LIN {X 0,Y 530.457,Z 403.715,A -85,B 0,C 180,E1 -4406.963,E2 -4406.963} C_VEL
LIN {X 0,Y 530.411,Z 405.124,A -85,B 0,C 180,E1 -4407.723,E2 -4407.723} C_VEL
LIN {X 0,Y 530.344,Z 406.736,A -85,B 0,C 180,E1 -4409.242,E2 -4409.242} C_VEL
LIN {X 0,Y 530.343,Z 406.953,A -85,B 0,C 180,E1 -4410.001,E2 -4410.001} C_VEL
LIN {X 0,Y 530.344,Z 406.734,A -85,B 0,C 180,E1 -4410.76,E2 -4410.76} C_VEL
LIN {X 0,Y 530.411,Z 405.118,A -85,B 0,C 180,E1 -4412.279,E2 -4412.279} C_VEL
LIN {X 0,Y 530.457,Z 403.708,A -85,B 0,C 180,E1 -4413.039,E2 -4413.039} C_VEL
LIN {X 0,Y 530.523,Z 400.73,A -85,B 0,C 180,E1 -4414.179,E2 -4414.179} C_VEL
LIN {X 0,Y 530.525,Z 396.658,A -85,B 0,C 180,E1 -4415.322,E2 -4415.322} C_VEL
LIN {X 0,Y 530.6,Z 390.764,A -85,B 0,C 180,E1 -4416.583,E2 -4416.583} C_VEL
LIN {X 0,Y 530.729,Z 383.488,A -85,B 0,C 180,E1 -4417.802,E2 -4417.802} C_VEL
LIN {X 0,Y 530.908,Z 374.945,A -85,B 0,C 180,E1 -4418.949,E2 -4418.949} C_VEL
LIN {X 0,Y 531.113,Z 365.145,A -85,B 0,C 180,E1 -4420.003,E2 -4420.003} C_VEL
LIN {X 0,Y 531.358,Z 354.095,A -85,B 0,C 180,E1 -4420.961,E2 -4420.961} C_VEL
LIN {X 0,Y 531.545,Z 343.017,A -85,B 0,C 180,E1 -4421.73,E2 -4421.73} C_VEL
LIN {X 0,Y 531.803,Z 330.634,A -85,B 0,C 180,E1 -4422.402,E2 -4422.402} C_VEL
LIN {X 0,Y 532.021,Z 317.664,A -85,B 0,C 180,E1 -4422.93,E2 -4422.93} C_VEL
LIN {X 0,Y 532.196,Z 304.731,A -85,B 0,C 180,E1 -4423.29,E2 -4423.29} C_VEL
LIN {X 0,Y 531.121,Z 293.757,A -85,B 0,C 180,E1 -4423.512,E2 -4423.512} C_VEL
LIN {X 0,Y 531.444,Z 271.801,A -85,B 0,C 180,E1 -4426.717,E2 -4426.717} C_VEL
LIN {X 0,Y 531.874,Z 250.491,A -85,B 0,C 180,E1 -4429.893,E2 -4429.893} C_VEL
LIN {X 0,Y 532.32,Z 231.821,A -85,B 0,C 180,E1 -4432.718,E2 -4432.718} C_VEL
LIN {X 0,Y 532.927,Z 210.283,A -85,B 0,C 180,E1 -4436.036,E2 -4436.036} C_VEL
LIN {X 0,Y 533.581,Z 192.22,A -85,B 0,C 180,E1 -4438.951,E2 -4438.951} C_VEL
LIN {X 0,Y 533.493,Z 188.442,A -85,B 0,C 180,E1 -4439.604,E2 -4439.604} C_VEL
LIN {X 0,Y 530.975,Z 177.349,A -85,B 0,C 180,E1 -4441.745,E2 -4441.745} C_VEL
LIN {X 0,Y 530.961,Z 177.352,A -85,B 0,C 180,E1 -4444.849,E2 -4444.849} C_VEL
LIN {X 0,Y 530.967,Z 177.345,A -85,B 0,C 180,E1 -4447.508,E2 -4447.508} C_VEL
LIN {X 0,Y 530.982,Z 177.347,A -85,B 0,C 180,E1 -4450.434,E2 -4450.434} C_VEL
LIN {X 0,Y 530.965,Z 177.345,A -85,B 0,C 180,E1 -4453.281,E2 -4453.281} C_VEL
LIN {X 0,Y 530.981,Z 177.348,A -85,B 0,C 180,E1 -4455.623,E2 -4455.623} C_VEL
LIN {X 0,Y 530.998,Z 177.341,A -85,B 0,C 180,E1 -4458.565,E2 -4458.565} C_VEL
LIN {X 0,Y 530.956,Z 177.347,A -85,B 0,C 180,E1 -4461.529,E2 -4461.529} C_VEL
LIN {X 0,Y 530.931,Z 177.355,A -85,B 0,C 180,E1 -4464.378,E2 -4464.378} C_VEL
LIN {X 0,Y 530.931,Z 177.42,A -85,B 0,C 180,E1 -4465.823,E2 -4465.823} C_VEL
LIN {X 0,Y 530.978,Z 185.304,A -85,B 0,C 180,E1 -4468.032,E2 -4468.032} C_VEL
LIN {X 0,Y 530.976,Z 194.876,A -85,B 0,C 180,E1 -4470.878,E2 -4470.878} C_VEL
LIN {X 0,Y 531.024,Z 203.845,A -85,B 0,C 180,E1 -4473.681,E2 -4473.681} C_VEL
LIN {X 0,Y 531.011,Z 212.797,A -85,B 0,C 180,E1 -4476.606,E2 -4476.606} C_VEL
LIN {X 0,Y 530.947,Z 221.236,A -85,B 0,C 180,E1 -4479.465,E2 -4479.465} C_VEL
LIN {X 0,Y 530.848,Z 229.893,A -85,B 0,C 180,E1 -4482.407,E2 -4482.407} C_VEL
LIN {X 0,Y 530.784,Z 238.562,A -85,B 0,C 180,E1 -4485.429,E2 -4485.429} C_VEL
LIN {X 0,Y 530.747,Z 241.715,A -85,B 0,C 180,E1 -4486.552,E2 -4486.552} C_VEL
LIN {X 0,Y 532.328,Z 250.665,A -85,B 0,C 180,E1 -4486.787,E2 -4486.787} C_VEL
LIN {X 0,Y 532.167,Z 262.9,A -85,B 0,C 180,E1 -4487.172,E2 -4487.172} C_VEL
LIN {X 0,Y 531.923,Z 274.906,A -85,B 0,C 180,E1 -4487.699,E2 -4487.699} C_VEL
LIN {X 0,Y 531.711,Z 286.037,A -85,B 0,C 180,E1 -4488.337,E2 -4488.337} C_VEL
LIN {X 0,Y 531.433,Z 297.075,A -85,B 0,C 180,E1 -4489.138,E2 -4489.138} C_VEL
LIN {X 0,Y 531.198,Z 307.619,A -85,B 0,C 180,E1 -4490.096,E2 -4490.096} C_VEL
LIN {X 0,Y 531.002,Z 316.164,A -85,B 0,C 180,E1 -4491.053,E2 -4491.053} C_VEL
LIN {X 0,Y 530.785,Z 324.463,A -85,B 0,C 180,E1 -4492.2,E2 -4492.2} C_VEL
LIN {X 0,Y 530.635,Z 331.357,A -85,B 0,C 180,E1 -4493.387,E2 -4493.387} C_VEL
LIN {X 0,Y 530.524,Z 337.207,A -85,B 0,C 180,E1 -4494.679,E2 -4494.679} C_VEL
LIN {X 0,Y 530.526,Z 341.159,A -85,B 0,C 180,E1 -4495.822,E2 -4495.822} C_VEL
LIN {X 0,Y 530.487,Z 344.081,A -85,B 0,C 180,E1 -4496.962,E2 -4496.962} C_VEL
LIN {X 0,Y 530.411,Z 345.518,A -85,B 0,C 180,E1 -4497.722,E2 -4497.722} C_VEL
LIN {X 0,Y 530.353,Z 347.118,A -85,B 0,C 180,E1 -4499.241,E2 -4499.241} C_VEL
LIN {X 0,Y 530.352,Z 347.354,A -85,B 0,C 180,E1 -4500,E2 -4500} C_VEL
LIN {X 0,Y 530.363,Z 346.589,A -85,B 0,C 180,E1 -4501.519,E2 -4501.519} C_VEL
LIN {X 0,Y 530.41,Z 345.633,A -85,B 0,C 180,E1 -4502.278,E2 -4502.278} C_VEL
LIN {X 0,Y 530.487,Z 344.255,A -85,B 0,C 180,E1 -4503.038,E2 -4503.038} C_VEL
LIN {X 0,Y 530.523,Z 341.398,A -85,B 0,C 180,E1 -4504.178,E2 -4504.178} C_VEL
LIN {X 0,Y 530.524,Z 337.512,A -85,B 0,C 180,E1 -4505.321,E2 -4505.321} C_VEL
LIN {X 0,Y 530.638,Z 331.546,A -85,B 0,C 180,E1 -4506.652,E2 -4506.652} C_VEL
LIN {X 0,Y 530.783,Z 324.976,A -85,B 0,C 180,E1 -4507.8,E2 -4507.8} C_VEL
LIN {X 0,Y 530.933,Z 316.768,A -85,B 0,C 180,E1 -4508.948,E2 -4508.948} C_VEL
LIN {X 0,Y 531.139,Z 308.382,A -85,B 0,C 180,E1 -4509.905,E2 -4509.905} C_VEL
LIN {X 0,Y 531.411,Z 298.042,A -85,B 0,C 180,E1 -4510.863,E2 -4510.863} C_VEL
LIN {X 0,Y 531.672,Z 286.414,A -85,B 0,C 180,E1 -4511.723,E2 -4511.723} C_VEL
LIN {X 0,Y 531.915,Z 274.672,A -85,B 0,C 180,E1 -4512.398,E2 -4512.398} C_VEL
LIN {X 0,Y 532.169,Z 262.615,A -85,B 0,C 180,E1 -4512.925,E2 -4512.925} C_VEL
LIN {X 0,Y 532.157,Z 249.903,A -85,B 0,C 180,E1 -4513.326,E2 -4513.326} C_VEL
LIN {X 0,Y 530.682,Z 241.294,A -85,B 0,C 180,E1 -4513.547,E2 -4513.547} C_VEL
LIN {X 0,Y 530.772,Z 232.779,A -85,B 0,C 180,E1 -4516.54,E2 -4516.54} C_VEL
LIN {X 0,Y 530.875,Z 224.872,A -85,B 0,C 180,E1 -4519.327,E2 -4519.327} C_VEL
LIN {X 0,Y 530.975,Z 215.665,A -85,B 0,C 180,E1 -4522.572,E2 -4522.572} C_VEL
LIN {X 0,Y 531.044,Z 207.423,A -85,B 0,C 180,E1 -4525.454,E2 -4525.454} C_VEL
LIN {X 0,Y 531.165,Z 198.965,A -85,B 0,C 180,E1 -4528.446,E2 -4528.446} C_VEL
LIN {X 0,Y 531.288,Z 191.5,A -85,B 0,C 180,E1 -4531.058,E2 -4531.058} C_VEL
LIN {X 0,Y 531.273,Z 183.807,A -85,B 0,C 180,E1 -4533.752,E2 -4533.752} C_VEL
LIN {X 0,Y 531.187,Z 178.509,A -85,B 0,C 180,E1 -4535.602,E2 -4535.602} C_VEL
LIN {X 0,Y 530.996,Z 177.346,A -85,B 0,C 180,E1 -4536.02,E2 -4536.02} C_VEL
LIN {X 0,Y 530.963,Z 177.349,A -85,B 0,C 180,E1 -4536.31,E2 -4536.31} C_VEL
LIN {X 0,Y 530.275,Z 177.434,A -85,B 0,C 180,E1 -4536.943,E2 -4536.943} C_VEL
LIN {X 0,Y 527.406,Z 177.792,A -85,B 0,C 180,E1 -4537.97,E2 -4537.97} C_VEL
LIN {X 0,Y 525.006,Z 178.088,A -85,B 0,C 180,E1 -4538.797,E2 -4538.797} C_VEL
LIN {X 0,Y 523.994,Z 178.217,A -85,B 0,C 180,E1 -4539.436,E2 -4539.436} C_VEL
LIN {X 0,Y 523.922,Z 178.22,A -85,B 0,C 180,E1 -4539.652,E2 -4539.652} C_VEL
LIN {X 0,Y 523.923,Z 178.225,A -85,B 0,C 180,E1 -4542.457,E2 -4542.457} C_VEL
LIN {X 0,Y 523.945,Z 178.218,A -85,B 0,C 180,E1 -4545.31,E2 -4545.31} C_VEL
LIN {X 0,Y 523.961,Z 178.218,A -85,B 0,C 180,E1 -4548.689,E2 -4548.689} C_VEL
LIN {X 0,Y 523.92,Z 178.224,A -85,B 0,C 180,E1 -4551.081,E2 -4551.081} C_VEL
LIN {X 0,Y 523.869,Z 178.234,A -85,B 0,C 180,E1 -4553.822,E2 -4553.822} C_VEL
LIN {X 0,Y 523.917,Z 178.224,A -85,B 0,C 180,E1 -4556.633,E2 -4556.633} C_VEL
LIN {X 0,Y 523.92,Z 178.223,A -85,B 0,C 180,E1 -4559.353,E2 -4559.353} C_VEL
LIN {X 0,Y 523.781,Z 178.245,A -85,B 0,C 180,E1 -4561.115,E2 -4561.115} C_VEL
LIN {X 0,Y 523.76,Z 181.958,A -85,B 0,C 180,E1 -4564.031,E2 -4564.031} C_VEL
LIN {X 0,Y 523.662,Z 185.872,A -85,B 0,C 180,E1 -4567.094,E2 -4567.094} C_VEL
LIN {X 0,Y 523.592,Z 190.074,A -85,B 0,C 180,E1 -4570.392,E2 -4570.392} C_VEL
LIN {X 0,Y 523.528,Z 193.22,A -85,B 0,C 180,E1 -4572.822,E2 -4572.822} C_VEL
LIN {X 0,Y 523.492,Z 197.581,A -85,B 0,C 180,E1 -4576.015,E2 -4576.015} C_VEL
LIN {X 0,Y 523.512,Z 202.047,A -85,B 0,C 180,E1 -4579.166,E2 -4579.166} C_VEL
LIN {X 0,Y 523.484,Z 206.049,A -85,B 0,C 180,E1 -4581.871,E2 -4581.871} C_VEL
LIN {X 0,Y 524.498,Z 212.037,A -85,B 0,C 180,E1 -4582.105,E2 -4582.105} C_VEL
LIN {X 0,Y 524.444,Z 221.603,A -85,B 0,C 180,E1 -4582.575,E2 -4582.575} C_VEL
LIN {X 0,Y 524.32,Z 230.114,A -85,B 0,C 180,E1 -4583.167,E2 -4583.167} C_VEL
LIN {X 0,Y 524.133,Z 237.545,A -85,B 0,C 180,E1 -4583.841,E2 -4583.841} C_VEL
LIN {X 0,Y 524.074,Z 243.948,A -85,B 0,C 180,E1 -4584.613,E2 -4584.613} C_VEL
LIN {X 0,Y 523.931,Z 250.016,A -85,B 0,C 180,E1 -4585.575,E2 -4585.575} C_VEL
LIN {X 0,Y 523.869,Z 254.451,A -85,B 0,C 180,E1 -4586.538,E2 -4586.538} C_VEL
LIN {X 0,Y 523.65,Z 258.123,A -85,B 0,C 180,E1 -4587.691,E2 -4587.691} C_VEL
LIN {X 0,Y 523.645,Z 259.678,A -85,B 0,C 180,E1 -4588.461,E2 -4588.461} C_VEL
LIN {X 0,Y 523.602,Z 260.61,A -85,B 0,C 180,E1 -4589.23,E2 -4589.23} C_VEL
LIN {X 0,Y 523.589,Z 260.941,A -85,B 0,C 180,E1 -4589.999,E2 -4589.999} C_VEL
LIN {X 0,Y 523.599,Z 260.684,A -85,B 0,C 180,E1 -4590.768,E2 -4590.768} C_VEL
LIN {X 0,Y 523.558,Z 259.84,A -85,B 0,C 180,E1 -4591.537,E2 -4591.537} C_VEL
LIN {X 0,Y 523.74,Z 257.352,A -85,B 0,C 180,E1 -4592.691,E2 -4592.691} C_VEL
LIN {X 0,Y 523.82,Z 253.258,A -85,B 0,C 180,E1 -4593.845,E2 -4593.845} C_VEL
LIN {X 0,Y 524.003,Z 248.362,A -85,B 0,C 180,E1 -4594.807,E2 -4594.807} C_VEL
LIN {X 0,Y 524.1,Z 241.688,A -85,B 0,C 180,E1 -4595.771,E2 -4595.771} C_VEL
LIN {X 0,Y 524.212,Z 234.727,A -85,B 0,C 180,E1 -4596.521,E2 -4596.521} C_VEL
LIN {X 0,Y 524.354,Z 226.524,A -85,B 0,C 180,E1 -4597.201,E2 -4597.201} C_VEL
LIN {X 0,Y 524.48,Z 218.274,A -85,B 0,C 180,E1 -4597.7,E2 -4597.7} C_VEL
LIN {X 0,Y 524.393,Z 210.728,A -85,B 0,C 180,E1 -4598.04,E2 -4598.04} C_VEL
LIN {X 0,Y 523.465,Z 206.053,A -85,B 0,C 180,E1 -4598.224,E2 -4598.224} C_VEL
LIN {X 0,Y 523.54,Z 201.101,A -85,B 0,C 180,E1 -4601.615,E2 -4601.615} C_VEL
LIN {X 0,Y 523.52,Z 196.503,A -85,B 0,C 180,E1 -4604.857,E2 -4604.857} C_VEL
LIN {X 0,Y 523.546,Z 192.298,A -85,B 0,C 180,E1 -4607.983,E2 -4607.983} C_VEL
LIN {X 0,Y 523.595,Z 189.157,A -85,B 0,C 180,E1 -4610.424,E2 -4610.424} C_VEL
LIN {X 0,Y 523.654,Z 186.02,A -85,B 0,C 180,E1 -4612.904,E2 -4612.904} C_VEL
LIN {X 0,Y 523.714,Z 182.822,A -85,B 0,C 180,E1 -4615.43,E2 -4615.43} C_VEL
LIN {X 0,Y 523.753,Z 179.451,A -85,B 0,C 180,E1 -4618.01,E2 -4618.01} C_VEL
LIN {X 0,Y 523.773,Z 178.296,A -85,B 0,C 180,E1 -4618.883,E2 -4618.883} C_VEL
LIN {X 0,Y 523.913,Z 178.227,A -85,B 0,C 180,E1 -4621.543,E2 -4621.543} C_VEL
LIN {X 0,Y 523.936,Z 178.218,A -85,B 0,C 180,E1 -4624.288,E2 -4624.288} C_VEL
LIN {X 0,Y 523.906,Z 178.226,A -85,B 0,C 180,E1 -4627.131,E2 -4627.131} C_VEL
LIN {X 0,Y 523.932,Z 178.218,A -85,B 0,C 180,E1 -4630.129,E2 -4630.129} C_VEL
LIN {X 0,Y 523.932,Z 178.218,A -85,B 0,C 180,E1 -4632.458,E2 -4632.458} C_VEL
LIN {X 0,Y 523.949,Z 178.22,A -85,B 0,C 180,E1 -4635.308,E2 -4635.308} C_VEL
LIN {X 0,Y 523.955,Z 178.221,A -85,B 0,C 180,E1 -4638.688,E2 -4638.688} C_VEL
LIN {X 0,Y 523.911,Z 178.22,A -85,B 0,C 180,E1 -4641.898,E2 -4641.898} C_VEL
LIN {X 0,Y 523.932,Z 178.221,A -85,B 0,C 180,E1 -4644.908,E2 -4644.908} C_VEL
LIN {X 0,Y 523.935,Z 178.217,A -85,B 0,C 180,E1 -4647.677,E2 -4647.677} C_VEL
LIN {X 0,Y 523.961,Z 178.217,A -85,B 0,C 180,E1 -4650.672,E2 -4650.672} C_VEL
LIN {X 0,Y 523.968,Z 178.216,A -85,B 0,C 180,E1 -4653.728,E2 -4653.728} C_VEL
LIN {X 0,Y 523.926,Z 178.224,A -85,B 0,C 180,E1 -4656.27,E2 -4656.27} C_VEL
LIN {X 0,Y 523.937,Z 178.216,A -85,B 0,C 180,E1 -4658.766,E2 -4658.766} C_VEL
LIN {X 0,Y 523.944,Z 178.216,A -85,B 0,C 180,E1 -4661.22,E2 -4661.22} C_VEL
LIN {X 0,Y 523.931,Z 178.225,A -85,B 0,C 180,E1 -4663.639,E2 -4663.639} C_VEL
LIN {X 0,Y 523.93,Z 178.22,A -85,B 0,C 180,E1 -4666.028,E2 -4666.028} C_VEL
LIN {X 0,Y 524,Z 178.208,A -85,B 0,C 180,E1 -4668.394,E2 -4668.394} C_VEL
LIN {X 0,Y 523.997,Z 178.215,A -85,B 0,C 180,E1 -4671.516,E2 -4671.516} C_VEL
LIN {X 0,Y 524.071,Z 178.2,A -85,B 0,C 180,E1 -4674.613,E2 -4674.613} C_VEL
LIN {X 0,Y 524.096,Z 178.198,A -85,B 0,C 180,E1 -4677.694,E2 -4677.694} C_VEL
LIN {X 0,Y 524.114,Z 178.197,A -85,B 0,C 180,E1 -4680.768,E2 -4680.768} C_VEL
LIN {X 0,Y 524.058,Z 178.206,A -85,B 0,C 180,E1 -4683.075,E2 -4683.075} C_VEL
LIN {X 0,Y 524.02,Z 178.207,A -85,B 0,C 180,E1 -4686.159,E2 -4686.159} C_VEL
LIN {X 0,Y 523.988,Z 178.218,A -85,B 0,C 180,E1 -4688.484,E2 -4688.484} C_VEL
LIN {X 0,Y 523.986,Z 178.212,A -85,B 0,C 180,E1 -4691.737,E2 -4691.737} C_VEL
LIN {X 0,Y 523.981,Z 178.212,A -85,B 0,C 180,E1 -4695.053,E2 -4695.053} C_VEL
LIN {X 0,Y 523.931,Z 178.222,A -85,B 0,C 180,E1 -4697.97,E2 -4697.97} C_VEL
LIN {X 0,Y 523.944,Z 178.22,A -85,B 0,C 180,E1 -4700.411,E2 -4700.411} C_VEL
LIN {X 0,Y 523.894,Z 178.223,A -85,B 0,C 180,E1 -4702.894,E2 -4702.894} C_VEL
LIN {X 0,Y 523.886,Z 178.227,A -85,B 0,C 180,E1 -4705.422,E2 -4705.422} C_VEL
LIN {X 0,Y 523.883,Z 178.229,A -85,B 0,C 180,E1 -4708.004,E2 -4708.004} C_VEL
LIN {X 0,Y 523.922,Z 178.22,A -85,B 0,C 180,E1 -4710.853,E2 -4710.853} C_VEL
LIN {X 0,Y 523.929,Z 178.221,A -85,B 0,C 180,E1 -4713.732,E2 -4713.732} C_VEL
LIN {X 0,Y 523.887,Z 178.224,A -85,B 0,C 180,E1 -4716.401,E2 -4716.401} C_VEL
LIN {X 0,Y 523.903,Z 178.23,A -85,B 0,C 180,E1 -4719.087,E2 -4719.087} C_VEL
LIN {X 0,Y 523.931,Z 178.219,A -85,B 0,C 180,E1 -4722.121,E2 -4722.121} C_VEL
LIN {X 0,Y 523.934,Z 178.221,A -85,B 0,C 180,E1 -4725.311,E2 -4725.311} C_VEL
LIN {X 0,Y 523.949,Z 178.22,A -85,B 0,C 180,E1 -4728.691,E2 -4728.691} C_VEL
LIN {X 0,Y 523.912,Z 178.225,A -85,B 0,C 180,E1 -4731.082,E2 -4731.082} C_VEL
LIN {X 0,Y 523.895,Z 178.224,A -85,B 0,C 180,E1 -4733.826,E2 -4733.826} C_VEL
LIN {X 0,Y 523.937,Z 178.224,A -85,B 0,C 180,E1 -4736.637,E2 -4736.637} C_VEL
LIN {X 0,Y 523.936,Z 178.33,A -85,B 0,C 180,E1 -4737.966,E2 -4737.966} C_VEL
LIN {X 0,Y 526.784,Z 190.799,A -85,B 0,C 180,E1 -4740.422,E2 -4740.422} C_VEL
LIN {X 0,Y 526.272,Z 203.612,A -85,B 0,C 180,E1 -4742.568,E2 -4742.568} C_VEL
LIN {X 0,Y 525.678,Z 221.266,A -85,B 0,C 180,E1 -4745.384,E2 -4745.384} C_VEL
LIN {X 0,Y 525.189,Z 239.466,A -85,B 0,C 180,E1 -4748.203,E2 -4748.203} C_VEL
LIN {X 0,Y 524.711,Z 259.403,A -85,B 0,C 180,E1 -4751.25,E2 -4751.25} C_VEL
LIN {X 0,Y 524.229,Z 280.571,A -85,B 0,C 180,E1 -4754.448,E2 -4754.448} C_VEL
LIN {X 0,Y 524.059,Z 293.373,A -85,B 0,C 180,E1 -4756.354,E2 -4756.354} C_VEL
LIN {X 0,Y 525.219,Z 305.411,A -85,B 0,C 180,E1 -4756.606,E2 -4756.606} C_VEL
LIN {X 0,Y 524.978,Z 318.332,A -85,B 0,C 180,E1 -4756.994,E2 -4756.994} C_VEL
LIN {X 0,Y 524.71,Z 330.841,A -85,B 0,C 180,E1 -4757.528,E2 -4757.528} C_VEL
LIN {X 0,Y 524.526,Z 342.894,A -85,B 0,C 180,E1 -4758.206,E2 -4758.206} C_VEL
LIN {X 0,Y 524.263,Z 353.816,A -85,B 0,C 180,E1 -4758.988,E2 -4758.988} C_VEL
LIN {X 0,Y 524.032,Z 364.766,A -85,B 0,C 180,E1 -4759.96,E2 -4759.96} C_VEL
LIN {X 0,Y 523.854,Z 373.636,A -85,B 0,C 180,E1 -4760.931,E2 -4760.931} C_VEL
LIN {X 0,Y 523.664,Z 382.289,A -85,B 0,C 180,E1 -4762.094,E2 -4762.094} C_VEL
LIN {X 0,Y 523.567,Z 388.184,A -85,B 0,C 180,E1 -4763.062,E2 -4763.062} C_VEL
LIN {X 0,Y 523.524,Z 393.933,A -85,B 0,C 180,E1 -4764.223,E2 -4764.223} C_VEL
LIN {X 0,Y 523.409,Z 398.424,A -85,B 0,C 180,E1 -4765.38,E2 -4765.38} C_VEL
LIN {X 0,Y 523.475,Z 400.815,A -85,B 0,C 180,E1 -4766.152,E2 -4766.152} C_VEL
LIN {X 0,Y 523.41,Z 402.733,A -85,B 0,C 180,E1 -4766.922,E2 -4766.922} C_VEL
LIN {X 0,Y 523.365,Z 404.183,A -85,B 0,C 180,E1 -4767.692,E2 -4767.692} C_VEL
LIN {X 0,Y 523.301,Z 405.828,A -85,B 0,C 180,E1 -4769.231,E2 -4769.231} C_VEL
LIN {X 0,Y 523.323,Z 406.053,A -85,B 0,C 180,E1 -4770.001,E2 -4770.001} C_VEL
LIN {X 0,Y 523.301,Z 405.828,A -85,B 0,C 180,E1 -4770.77,E2 -4770.77} C_VEL
LIN {X 0,Y 523.365,Z 404.178,A -85,B 0,C 180,E1 -4772.31,E2 -4772.31} C_VEL
LIN {X 0,Y 523.411,Z 402.719,A -85,B 0,C 180,E1 -4773.08,E2 -4773.08} C_VEL
LIN {X 0,Y 523.475,Z 399.687,A -85,B 0,C 180,E1 -4774.236,E2 -4774.236} C_VEL
LIN {X 0,Y 523.477,Z 395.565,A -85,B 0,C 180,E1 -4775.394,E2 -4775.394} C_VEL
LIN {X 0,Y 523.561,Z 389.907,A -85,B 0,C 180,E1 -4776.616,E2 -4776.616} C_VEL
LIN {X 0,Y 523.666,Z 382.263,A -85,B 0,C 180,E1 -4777.908,E2 -4777.908} C_VEL
LIN {X 0,Y 523.855,Z 373.634,A -85,B 0,C 180,E1 -4779.071,E2 -4779.071} C_VEL
LIN {X 0,Y 524.066,Z 363.735,A -85,B 0,C 180,E1 -4780.139,E2 -4780.139} C_VEL
LIN {X 0,Y 524.314,Z 352.589,A -85,B 0,C 180,E1 -4781.11,E2 -4781.11} C_VEL
LIN {X 0,Y 524.462,Z 341.902,A -85,B 0,C 180,E1 -4781.856,E2 -4781.856} C_VEL
LIN {X 0,Y 524.742,Z 330.812,A -85,B 0,C 180,E1 -4782.473,E2 -4782.473} C_VEL
LIN {X 0,Y 524.991,Z 318.292,A -85,B 0,C 180,E1 -4783.008,E2 -4783.008} C_VEL
LIN {X 0,Y 525.195,Z 305.317,A -85,B 0,C 180,E1 -4783.396,E2 -4783.396} C_VEL
LIN {X 0,Y 524.059,Z 293.335,A -85,B 0,C 180,E1 -4783.648,E2 -4783.648} C_VEL
LIN {X 0,Y 524.395,Z 272.602,A -85,B 0,C 180,E1 -4786.748,E2 -4786.748} C_VEL
LIN {X 0,Y 524.836,Z 252.725,A -85,B 0,C 180,E1 -4789.763,E2 -4789.763} C_VEL
LIN {X 0,Y 525.28,Z 236.105,A -85,B 0,C 180,E1 -4792.313,E2 -4792.313} C_VEL
LIN {X 0,Y 525.804,Z 216.755,A -85,B 0,C 180,E1 -4795.324,E2 -4795.324} C_VEL
LIN {X 0,Y 526.522,Z 198.672,A -85,B 0,C 180,E1 -4798.24,E2 -4798.24} C_VEL
LIN {X 0,Y 526.763,Z 190.817,A -85,B 0,C 180,E1 -4799.581,E2 -4799.581} C_VEL
LIN {X 0,Y 523.929,Z 178.227,A -85,B 0,C 180,E1 -4802.056,E2 -4802.056} C_VEL
LIN {X 0,Y 523.921,Z 178.228,A -85,B 0,C 180,E1 -4805.088,E2 -4805.088} C_VEL
LIN {X 0,Y 523.917,Z 178.225,A -85,B 0,C 180,E1 -4808.103,E2 -4808.103} C_VEL
LIN {X 0,Y 523.961,Z 178.216,A -85,B 0,C 180,E1 -4811.311,E2 -4811.311} C_VEL
LIN {X 0,Y 523.947,Z 178.218,A -85,B 0,C 180,E1 -4814.69,E2 -4814.69} C_VEL
LIN {X 0,Y 523.956,Z 178.219,A -85,B 0,C 180,E1 -4817.881,E2 -4817.881} C_VEL
LIN {X 0,Y 523.916,Z 178.228,A -85,B 0,C 180,E1 -4820.915,E2 -4820.915} C_VEL
LIN {X 0,Y 523.881,Z 178.229,A -85,B 0,C 180,E1 -4823.824,E2 -4823.824} C_VEL
LIN {X 0,Y 523.885,Z 178.311,A -85,B 0,C 180,E1 -4825.706,E2 -4825.706} C_VEL
LIN {X 0,Y 523.995,Z 185.239,A -85,B 0,C 180,E1 -4827.67,E2 -4827.67} C_VEL
LIN {X 0,Y 523.965,Z 195.34,A -85,B 0,C 180,E1 -4830.676,E2 -4830.676} C_VEL
LIN {X 0,Y 523.997,Z 205.047,A -85,B 0,C 180,E1 -4833.73,E2 -4833.73} C_VEL
LIN {X 0,Y 523.959,Z 213.975,A -85,B 0,C 180,E1 -4836.691,E2 -4836.691} C_VEL
LIN {X 0,Y 523.918,Z 221.424,A -85,B 0,C 180,E1 -4839.177,E2 -4839.177} C_VEL
LIN {X 0,Y 523.845,Z 229.751,A -85,B 0,C 180,E1 -4842.027,E2 -4842.027} C_VEL
LIN {X 0,Y 523.748,Z 238.929,A -85,B 0,C 180,E1 -4845.229,E2 -4845.229} C_VEL
LIN {X 0,Y 523.725,Z 242.375,A -85,B 0,C 180,E1 -4846.381,E2 -4846.381} C_VEL
LIN {X 0,Y 525.414,Z 251.672,A -85,B 0,C 180,E1 -4846.635,E2 -4846.635} C_VEL
LIN {X 0,Y 525.228,Z 264.272,A -85,B 0,C 180,E1 -4847.048,E2 -4847.048} C_VEL
LIN {X 0,Y 524.928,Z 276.955,A -85,B 0,C 180,E1 -4847.63,E2 -4847.63} C_VEL
LIN {X 0,Y 524.746,Z 288.15,A -85,B 0,C 180,E1 -4848.306,E2 -4848.306} C_VEL
LIN {X 0,Y 524.402,Z 299.64,A -85,B 0,C 180,E1 -4849.186,E2 -4849.186} C_VEL
LIN {X 0,Y 524.151,Z 309.76,A -85,B 0,C 180,E1 -4850.157,E2 -4850.157} C_VEL
LIN {X 0,Y 523.954,Z 317.987,A -85,B 0,C 180,E1 -4851.126,E2 -4851.126} C_VEL
LIN {X 0,Y 523.729,Z 326.026,A -85,B 0,C 180,E1 -4852.288,E2 -4852.288} C_VEL
LIN {X 0,Y 523.596,Z 331.989,A -85,B 0,C 180,E1 -4853.352,E2 -4853.352} C_VEL
LIN {X 0,Y 523.463,Z 337.583,A -85,B 0,C 180,E1 -4854.607,E2 -4854.607} C_VEL
LIN {X 0,Y 523.454,Z 341.544,A -85,B 0,C 180,E1 -4855.765,E2 -4855.765} C_VEL
LIN {X 0,Y 523.424,Z 344.47,A -85,B 0,C 180,E1 -4856.921,E2 -4856.921} C_VEL
LIN {X 0,Y 523.336,Z 345.907,A -85,B 0,C 180,E1 -4857.691,E2 -4857.691} C_VEL
LIN {X 0,Y 523.265,Z 347.508,A -85,B 0,C 180,E1 -4859.23,E2 -4859.23} C_VEL
LIN {X 0,Y 523.263,Z 347.74,A -85,B 0,C 180,E1 -4860,E2 -4860} C_VEL
LIN {X 0,Y 523.277,Z 346.968,A -85,B 0,C 180,E1 -4861.539,E2 -4861.539} C_VEL
LIN {X 0,Y 523.336,Z 346.001,A -85,B 0,C 180,E1 -4862.309,E2 -4862.309} C_VEL
LIN {X 0,Y 523.424,Z 344.617,A -85,B 0,C 180,E1 -4863.079,E2 -4863.079} C_VEL
LIN {X 0,Y 523.447,Z 341.746,A -85,B 0,C 180,E1 -4864.235,E2 -4864.235} C_VEL
LIN {X 0,Y 523.463,Z 337.843,A -85,B 0,C 180,E1 -4865.393,E2 -4865.393} C_VEL
LIN {X 0,Y 523.571,Z 332.233,A -85,B 0,C 180,E1 -4866.665,E2 -4866.665} C_VEL
LIN {X 0,Y 523.758,Z 325.253,A -85,B 0,C 180,E1 -4867.906,E2 -4867.906} C_VEL
LIN {X 0,Y 523.918,Z 317.024,A -85,B 0,C 180,E1 -4869.069,E2 -4869.069} C_VEL
LIN {X 0,Y 524.136,Z 308.608,A -85,B 0,C 180,E1 -4870.039,E2 -4870.039} C_VEL
LIN {X 0,Y 524.427,Z 298.234,A -85,B 0,C 180,E1 -4871.009,E2 -4871.009} C_VEL
LIN {X 0,Y 524.709,Z 287.137,A -85,B 0,C 180,E1 -4871.843,E2 -4871.843} C_VEL
LIN {X 0,Y 524.974,Z 274.789,A -85,B 0,C 180,E1 -4872.565,E2 -4872.565} C_VEL
LIN {X 0,Y 525.245,Z 262.698,A -85,B 0,C 180,E1 -4873.099,E2 -4873.099} C_VEL
LIN {X 0,Y 525.273,Z 250.855,A -85,B 0,C 180,E1 -4873.48,E2 -4873.48} C_VEL
LIN {X 0,Y 523.619,Z 241.62,A -85,B 0,C 180,E1 -4873.733,E2 -4873.733} C_VEL
LIN {X 0,Y 523.751,Z 233.011,A -85,B 0,C 180,E1 -4876.768,E2 -4876.768} C_VEL
LIN {X 0,Y 523.844,Z 224.99,A -85,B 0,C 180,E1 -4879.597,E2 -4879.597} C_VEL
LIN {X 0,Y 523.926,Z 217.502,A -85,B 0,C 180,E1 -4882.244,E2 -4882.244} C_VEL
LIN {X 0,Y 524.014,Z 208.556,A -85,B 0,C 180,E1 -4885.416,E2 -4885.416} C_VEL
LIN {X 0,Y 524.155,Z 200.11,A -85,B 0,C 180,E1 -4888.424,E2 -4888.424} C_VEL
LIN {X 0,Y 524.277,Z 191.31,A -85,B 0,C 180,E1 -4891.52,E2 -4891.52} C_VEL
LIN {X 0,Y 524.32,Z 182.231,A -85,B 0,C 180,E1 -4894.703,E2 -4894.703} C_VEL
LIN {X 0,Y 523.927,Z 178.226,A -85,B 0,C 180,E1 -4896.173,E2 -4896.173} C_VEL
LIN {X 0,Y 523.924,Z 178.223,A -85,B 0,C 180,E1 -4899.085,E2 -4899.085} C_VEL
LIN {X 0,Y 523.922,Z 178.22,A -85,B 0,C 180,E1 -4899.652,E2 -4899.652} C_VEL
LIN {X 0,Y 523.278,Z 178.303,A -85,B 0,C 180,E1 -4900.295,E2 -4900.295} C_VEL
LIN {X 0,Y 520.422,Z 178.663,A -85,B 0,C 180,E1 -4901.337,E2 -4901.337} C_VEL
LIN {X 0,Y 517.988,Z 178.967,A -85,B 0,C 180,E1 -4902.176,E2 -4902.176} C_VEL
LIN {X 0,Y 516.938,Z 179.096,A -85,B 0,C 180,E1 -4902.824,E2 -4902.824} C_VEL
LIN {X 0,Y 516.851,Z 179.104,A -85,B 0,C 180,E1 -4903.044,E2 -4903.044} C_VEL
LIN {X 0,Y 516.887,Z 179.101,A -85,B 0,C 180,E1 -4906.107,E2 -4906.107} C_VEL
LIN {X 0,Y 516.919,Z 179.094,A -85,B 0,C 180,E1 -4908.398,E2 -4908.398} C_VEL
LIN {X 0,Y 516.882,Z 179.1,A -85,B 0,C 180,E1 -4911.283,E2 -4911.283} C_VEL
LIN {X 0,Y 516.857,Z 179.103,A -85,B 0,C 180,E1 -4914.672,E2 -4914.672} C_VEL
LIN {X 0,Y 516.9,Z 179.099,A -85,B 0,C 180,E1 -4917.457,E2 -4917.457} C_VEL
LIN {X 0,Y 516.833,Z 179.106,A -85,B 0,C 180,E1 -4919.792,E2 -4919.792} C_VEL
LIN {X 0,Y 516.778,Z 179.117,A -85,B 0,C 180,E1 -4920.686,E2 -4920.686} C_VEL
LIN {X 0,Y 516.695,Z 179.578,A -85,B 0,C 180,E1 -4921.57,E2 -4921.57} C_VEL
LIN {X 0,Y 516.688,Z 182.944,A -85,B 0,C 180,E1 -4924.197,E2 -4924.197} C_VEL
LIN {X 0,Y 516.592,Z 186.215,A -85,B 0,C 180,E1 -4926.762,E2 -4926.762} C_VEL
LIN {X 0,Y 516.546,Z 190.463,A -85,B 0,C 180,E1 -4930.113,E2 -4930.113} C_VEL
LIN {X 0,Y 516.47,Z 193.618,A -85,B 0,C 180,E1 -4932.579,E2 -4932.579} C_VEL
LIN {X 0,Y 516.435,Z 197.985,A -85,B 0,C 180,E1 -4935.82,E2 -4935.82} C_VEL
LIN {X 0,Y 516.448,Z 202.522,A -85,B 0,C 180,E1 -4939.016,E2 -4939.016} C_VEL
LIN {X 0,Y 516.432,Z 206.68,A -85,B 0,C 180,E1 -4941.71,E2 -4941.71} C_VEL
LIN {X 0,Y 517.581,Z 212.783,A -85,B 0,C 180,E1 -4941.95,E2 -4941.95} C_VEL
LIN {X 0,Y 517.544,Z 221.422,A -85,B 0,C 180,E1 -4942.362,E2 -4942.362} C_VEL
LIN {X 0,Y 517.448,Z 228.989,A -85,B 0,C 180,E1 -4942.862,E2 -4942.862} C_VEL
LIN {X 0,Y 517.254,Z 236.031,A -85,B 0,C 180,E1 -4943.465,E2 -4943.465} C_VEL
LIN {X 0,Y 517.216,Z 242.28,A -85,B 0,C 180,E1 -4944.15,E2 -4944.15} C_VEL
LIN {X 0,Y 517.098,Z 247.888,A -85,B 0,C 180,E1 -4944.931,E2 -4944.931} C_VEL
LIN {X 0,Y 516.927,Z 252.223,A -85,B 0,C 180,E1 -4945.711,E2 -4945.711} C_VEL
LIN {X 0,Y 516.797,Z 256.971,A -85,B 0,C 180,E1 -4946.881,E2 -4946.881} C_VEL
LIN {X 0,Y 516.642,Z 259.177,A -85,B 0,C 180,E1 -4947.66,E2 -4947.66} C_VEL
LIN {X 0,Y 516.639,Z 260.689,A -85,B 0,C 180,E1 -4948.44,E2 -4948.44} C_VEL
LIN {X 0,Y 516.589,Z 261.594,A -85,B 0,C 180,E1 -4949.219,E2 -4949.219} C_VEL
LIN {X 0,Y 516.573,Z 261.913,A -85,B 0,C 180,E1 -4949.999,E2 -4949.999} C_VEL
LIN {X 0,Y 516.585,Z 261.663,A -85,B 0,C 180,E1 -4950.779,E2 -4950.779} C_VEL
LIN {X 0,Y 516.536,Z 260.845,A -85,B 0,C 180,E1 -4951.558,E2 -4951.558} C_VEL
LIN {X 0,Y 516.741,Z 258.417,A -85,B 0,C 180,E1 -4952.727,E2 -4952.727} C_VEL
LIN {X 0,Y 516.83,Z 254.415,A -85,B 0,C 180,E1 -4953.898,E2 -4953.898} C_VEL
LIN {X 0,Y 517.055,Z 249.608,A -85,B 0,C 180,E1 -4954.872,E2 -4954.872} C_VEL
LIN {X 0,Y 517.171,Z 243.057,A -85,B 0,C 180,E1 -4955.849,E2 -4955.849} C_VEL
LIN {X 0,Y 517.279,Z 235.974,A -85,B 0,C 180,E1 -4956.631,E2 -4956.631} C_VEL
LIN {X 0,Y 517.424,Z 228.437,A -85,B 0,C 180,E1 -4957.273,E2 -4957.273} C_VEL
LIN {X 0,Y 517.554,Z 220.037,A -85,B 0,C 180,E1 -4957.803,E2 -4957.803} C_VEL
LIN {X 0,Y 517.431,Z 211.437,A -85,B 0,C 180,E1 -4958.198,E2 -4958.198} C_VEL
LIN {X 0,Y 516.406,Z 206.524,A -85,B 0,C 180,E1 -4958.412,E2 -4958.412} C_VEL
LIN {X 0,Y 516.472,Z 201.535,A -85,B 0,C 180,E1 -4961.777,E2 -4961.777} C_VEL
LIN {X 0,Y 516.455,Z 196.997,A -85,B 0,C 180,E1 -4964.983,E2 -4964.983} C_VEL
LIN {X 0,Y 516.482,Z 192.698,A -85,B 0,C 180,E1 -4968.237,E2 -4968.237} C_VEL
LIN {X 0,Y 516.529,Z 189.542,A -85,B 0,C 180,E1 -4970.716,E2 -4970.716} C_VEL
LIN {X 0,Y 516.587,Z 186.366,A -85,B 0,C 180,E1 -4973.236,E2 -4973.236} C_VEL
LIN {X 0,Y 516.683,Z 182.679,A -85,B 0,C 180,E1 -4976.137,E2 -4976.137} C_VEL
LIN {X 0,Y 516.693,Z 179.702,A -85,B 0,C 180,E1 -4978.427,E2 -4978.427} C_VEL
LIN {X 0,Y 516.817,Z 179.112,A -85,B 0,C 180,E1 -4979.505,E2 -4979.505} C_VEL
LIN {X 0,Y 516.869,Z 179.101,A -85,B 0,C 180,E1 -4982.024,E2 -4982.024} C_VEL
LIN {X 0,Y 516.887,Z 179.097,A -85,B 0,C 180,E1 -4984.823,E2 -4984.823} C_VEL
LIN {X 0,Y 516.876,Z 179.099,A -85,B 0,C 180,E1 -4987.942,E2 -4987.942} C_VEL
LIN {X 0,Y 516.879,Z 179.099,A -85,B 0,C 180,E1 -4990.74,E2 -4990.74} C_VEL
LIN {X 0,Y 516.898,Z 179.098,A -85,B 0,C 180,E1 -4992.828,E2 -4992.828} C_VEL
LIN {X 0,Y 516.916,Z 179.099,A -85,B 0,C 180,E1 -4995.009,E2 -4995.009} C_VEL
LIN {X 0,Y 516.91,Z 179.095,A -85,B 0,C 180,E1 -4998.397,E2 -4998.397} C_VEL
LIN {X 0,Y 516.876,Z 179.098,A -85,B 0,C 180,E1 -5001.283,E2 -5001.283} C_VEL
LIN {X 0,Y 516.883,Z 179.099,A -85,B 0,C 180,E1 -5004.22,E2 -5004.22} C_VEL
LIN {X 0,Y 516.89,Z 179.096,A -85,B 0,C 180,E1 -5007.052,E2 -5007.052} C_VEL
LIN {X 0,Y 516.893,Z 179.096,A -85,B 0,C 180,E1 -5009.796,E2 -5009.796} C_VEL
LIN {X 0,Y 516.921,Z 179.096,A -85,B 0,C 180,E1 -5012.467,E2 -5012.467} C_VEL
LIN {X 0,Y 516.902,Z 179.09,A -85,B 0,C 180,E1 -5015.071,E2 -5015.071} C_VEL
LIN {X 0,Y 516.877,Z 179.097,A -85,B 0,C 180,E1 -5018.462,E2 -5018.462} C_VEL
LIN {X 0,Y 516.894,Z 179.093,A -85,B 0,C 180,E1 -5020.954,E2 -5020.954} C_VEL
LIN {X 0,Y 516.908,Z 179.097,A -85,B 0,C 180,E1 -5023.41,E2 -5023.41} C_VEL
LIN {X 0,Y 516.886,Z 179.1,A -85,B 0,C 180,E1 -5025.833,E2 -5025.833} C_VEL
LIN {X 0,Y 516.946,Z 179.09,A -85,B 0,C 180,E1 -5029.028,E2 -5029.028} C_VEL
LIN {X 0,Y 516.968,Z 179.085,A -85,B 0,C 180,E1 -5032.187,E2 -5032.187} C_VEL
LIN {X 0,Y 517.018,Z 179.078,A -85,B 0,C 180,E1 -5034.54,E2 -5034.54} C_VEL
LIN {X 0,Y 517.068,Z 179.074,A -85,B 0,C 180,E1 -5037.663,E2 -5037.663} C_VEL
LIN {X 0,Y 517.084,Z 179.073,A -85,B 0,C 180,E1 -5040.779,E2 -5040.779} C_VEL
LIN {X 0,Y 516.998,Z 179.085,A -85,B 0,C 180,E1 -5043.117,E2 -5043.117} C_VEL
LIN {X 0,Y 516.986,Z 179.084,A -85,B 0,C 180,E1 -5046.243,E2 -5046.243} C_VEL
LIN {X 0,Y 516.952,Z 179.092,A -85,B 0,C 180,E1 -5048.601,E2 -5048.601} C_VEL
LIN {X 0,Y 516.939,Z 179.09,A -85,B 0,C 180,E1 -5051.807,E2 -5051.807} C_VEL
LIN {X 0,Y 516.932,Z 179.09,A -85,B 0,C 180,E1 -5055.147,E2 -5055.147} C_VEL
LIN {X 0,Y 516.899,Z 179.1,A -85,B 0,C 180,E1 -5058.223,E2 -5058.223} C_VEL
LIN {X 0,Y 516.891,Z 179.096,A -85,B 0,C 180,E1 -5060.702,E2 -5060.702} C_VEL
LIN {X 0,Y 516.872,Z 179.104,A -85,B 0,C 180,E1 -5064.074,E2 -5064.074} C_VEL
LIN {X 0,Y 516.824,Z 179.104,A -85,B 0,C 180,E1 -5066.663,E2 -5066.663} C_VEL
LIN {X 0,Y 516.873,Z 179.105,A -85,B 0,C 180,E1 -5069.519,E2 -5069.519} C_VEL
LIN {X 0,Y 516.884,Z 179.096,A -85,B 0,C 180,E1 -5072.544,E2 -5072.544} C_VEL
LIN {X 0,Y 516.85,Z 179.106,A -85,B 0,C 180,E1 -5075.33,E2 -5075.33} C_VEL
LIN {X 0,Y 516.868,Z 179.1,A -85,B 0,C 180,E1 -5077.943,E2 -5077.943} C_VEL
LIN {X 0,Y 516.855,Z 179.1,A -85,B 0,C 180,E1 -5080.745,E2 -5080.745} C_VEL
LIN {X 0,Y 516.85,Z 179.107,A -85,B 0,C 180,E1 -5082.835,E2 -5082.835} C_VEL
LIN {X 0,Y 516.887,Z 179.102,A -85,B 0,C 180,E1 -5085.008,E2 -5085.008} C_VEL
LIN {X 0,Y 516.906,Z 179.093,A -85,B 0,C 180,E1 -5088.4,E2 -5088.4} C_VEL
LIN {X 0,Y 516.875,Z 179.1,A -85,B 0,C 180,E1 -5091.285,E2 -5091.285} C_VEL
LIN {X 0,Y 516.866,Z 179.104,A -85,B 0,C 180,E1 -5094.221,E2 -5094.221} C_VEL
LIN {X 0,Y 516.89,Z 179.102,A -85,B 0,C 180,E1 -5097.054,E2 -5097.054} C_VEL
LIN {X 0,Y 516.924,Z 179.308,A -85,B 0,C 180,E1 -5097.667,E2 -5097.667} C_VEL
LIN {X 0,Y 519.713,Z 191.425,A -85,B 0,C 180,E1 -5100.117,E2 -5100.117} C_VEL
LIN {X 0,Y 519.928,Z 194.44,A -85,B 0,C 180,E1 -5100.661,E2 -5100.661} C_VEL
LIN {X 0,Y 519.174,Z 211.183,A -85,B 0,C 180,E1 -5103.468,E2 -5103.468} C_VEL
LIN {X 0,Y 518.504,Z 231.074,A -85,B 0,C 180,E1 -5106.644,E2 -5106.644} C_VEL
LIN {X 0,Y 517.919,Z 251.213,A -85,B 0,C 180,E1 -5109.787,E2 -5109.787} C_VEL
LIN {X 0,Y 517.462,Z 269.487,A -85,B 0,C 180,E1 -5112.616,E2 -5112.616} C_VEL
LIN {X 0,Y 517.007,Z 291.696,A -85,B 0,C 180,E1 -5116.039,E2 -5116.039} C_VEL
LIN {X 0,Y 517.017,Z 292.989,A -85,B 0,C 180,E1 -5116.214,E2 -5116.214} C_VEL
LIN {X 0,Y 518.131,Z 304.369,A -85,B 0,C 180,E1 -5116.457,E2 -5116.457} C_VEL
LIN {X 0,Y 517.971,Z 317.598,A -85,B 0,C 180,E1 -5116.865,E2 -5116.865} C_VEL
LIN {X 0,Y 517.654,Z 331.009,A -85,B 0,C 180,E1 -5117.455,E2 -5117.455} C_VEL
LIN {X 0,Y 517.447,Z 342.941,A -85,B 0,C 180,E1 -5118.154,E2 -5118.154} C_VEL
LIN {X 0,Y 517.181,Z 353.512,A -85,B 0,C 180,E1 -5118.935,E2 -5118.935} C_VEL
LIN {X 0,Y 516.995,Z 363.364,A -85,B 0,C 180,E1 -5119.822,E2 -5119.822} C_VEL
LIN {X 0,Y 516.776,Z 372.309,A -85,B 0,C 180,E1 -5120.806,E2 -5120.806} C_VEL
LIN {X 0,Y 516.62,Z 381.059,A -85,B 0,C 180,E1 -5121.986,E2 -5121.986} C_VEL
LIN {X 0,Y 516.488,Z 388.188,A -85,B 0,C 180,E1 -5123.185,E2 -5123.185} C_VEL
LIN {X 0,Y 516.424,Z 394.462,A -85,B 0,C 180,E1 -5124.535,E2 -5124.535} C_VEL
LIN {X 0,Y 516.429,Z 398.637,A -85,B 0,C 180,E1 -5125.709,E2 -5125.709} C_VEL
LIN {X 0,Y 516.368,Z 401.715,A -85,B 0,C 180,E1 -5126.88,E2 -5126.88} C_VEL
LIN {X 0,Y 516.326,Z 403.181,A -85,B 0,C 180,E1 -5127.661,E2 -5127.661} C_VEL
LIN {X 0,Y 516.281,Z 404.224,A -85,B 0,C 180,E1 -5128.441,E2 -5128.441} C_VEL
LIN {X 0,Y 516.285,Z 404.855,A -85,B 0,C 180,E1 -5129.221,E2 -5129.221} C_VEL
LIN {X 0,Y 516.303,Z 405.08,A -85,B 0,C 180,E1 -5130.001,E2 -5130.001} C_VEL
LIN {X 0,Y 516.285,Z 404.839,A -85,B 0,C 180,E1 -5130.781,E2 -5130.781} C_VEL
LIN {X 0,Y 516.325,Z 403.189,A -85,B 0,C 180,E1 -5132.341,E2 -5132.341} C_VEL
LIN {X 0,Y 516.37,Z 401.69,A -85,B 0,C 180,E1 -5133.122,E2 -5133.122} C_VEL
LIN {X 0,Y 516.43,Z 398.631,A -85,B 0,C 180,E1 -5134.293,E2 -5134.293} C_VEL
LIN {X 0,Y 516.424,Z 394.468,A -85,B 0,C 180,E1 -5135.467,E2 -5135.467} C_VEL
LIN {X 0,Y 516.504,Z 388.1,A -85,B 0,C 180,E1 -5136.829,E2 -5136.829} C_VEL
LIN {X 0,Y 516.622,Z 381.032,A -85,B 0,C 180,E1 -5138.016,E2 -5138.016} C_VEL
LIN {X 0,Y 516.778,Z 372.304,A -85,B 0,C 180,E1 -5139.196,E2 -5139.196} C_VEL
LIN {X 0,Y 517.027,Z 362.324,A -85,B 0,C 180,E1 -5140.278,E2 -5140.278} C_VEL
LIN {X 0,Y 517.236,Z 352.293,A -85,B 0,C 180,E1 -5141.165,E2 -5141.165} C_VEL
LIN {X 0,Y 517.379,Z 342.033,A -85,B 0,C 180,E1 -5141.907,E2 -5141.907} C_VEL
LIN {X 0,Y 517.7,Z 330.982,A -85,B 0,C 180,E1 -5142.546,E2 -5142.546} C_VEL
LIN {X 0,Y 517.965,Z 317.552,A -85,B 0,C 180,E1 -5143.137,E2 -5143.137} C_VEL
LIN {X 0,Y 518.158,Z 304.274,A -85,B 0,C 180,E1 -5143.544,E2 -5143.544} C_VEL
LIN {X 0,Y 517.038,Z 293.73,A -85,B 0,C 180,E1 -5143.775,E2 -5143.775} C_VEL
LIN {X 0,Y 517.013,Z 292.685,A -85,B 0,C 180,E1 -5143.813,E2 -5143.813} C_VEL
LIN {X 0,Y 517.405,Z 270.727,A -85,B 0,C 180,E1 -5147.184,E2 -5147.184} C_VEL
LIN {X 0,Y 517.987,Z 249.55,A -85,B 0,C 180,E1 -5150.472,E2 -5150.472} C_VEL
LIN {X 0,Y 518.6,Z 228.4,A -85,B 0,C 180,E1 -5153.777,E2 -5153.777} C_VEL
LIN {X 0,Y 519.306,Z 208.4,A -85,B 0,C 180,E1 -5156.987,E2 -5156.987} C_VEL
LIN {X 0,Y 519.953,Z 193.166,A -85,B 0,C 180,E1 -5159.562,E2 -5159.562} C_VEL
LIN {X 0,Y 517.537,Z 181.932,A -85,B 0,C 180,E1 -5161.78,E2 -5161.78} C_VEL
LIN {X 0,Y 516.884,Z 179.105,A -85,B 0,C 180,E1 -5162.381,E2 -5162.381} C_VEL
LIN {X 0,Y 516.864,Z 179.106,A -85,B 0,C 180,E1 -5165.329,E2 -5165.329} C_VEL
LIN {X 0,Y 516.882,Z 179.1,A -85,B 0,C 180,E1 -5167.943,E2 -5167.943} C_VEL
LIN {X 0,Y 516.888,Z 179.099,A -85,B 0,C 180,E1 -5170.742,E2 -5170.742} C_VEL
LIN {X 0,Y 516.887,Z 179.098,A -85,B 0,C 180,E1 -5172.832,E2 -5172.832} C_VEL
LIN {X 0,Y 516.9,Z 179.097,A -85,B 0,C 180,E1 -5175.007,E2 -5175.007} C_VEL
LIN {X 0,Y 516.918,Z 179.095,A -85,B 0,C 180,E1 -5178.399,E2 -5178.399} C_VEL
LIN {X 0,Y 516.88,Z 179.103,A -85,B 0,C 180,E1 -5181.284,E2 -5181.284} C_VEL
LIN {X 0,Y 516.818,Z 179.112,A -85,B 0,C 180,E1 -5184.215,E2 -5184.215} C_VEL
LIN {X 0,Y 516.866,Z 179.228,A -85,B 0,C 180,E1 -5185.58,E2 -5185.58} C_VEL
LIN {X 0,Y 517.016,Z 185.713,A -85,B 0,C 180,E1 -5187.437,E2 -5187.437} C_VEL
LIN {X 0,Y 516.967,Z 195.835,A -85,B 0,C 180,E1 -5190.467,E2 -5190.467} C_VEL
LIN {X 0,Y 516.979,Z 204.943,A -85,B 0,C 180,E1 -5193.345,E2 -5193.345} C_VEL
LIN {X 0,Y 516.966,Z 214.091,A -85,B 0,C 180,E1 -5196.357,E2 -5196.357} C_VEL
LIN {X 0,Y 516.884,Z 222.795,A -85,B 0,C 180,E1 -5199.297,E2 -5199.297} C_VEL
LIN {X 0,Y 516.795,Z 231.141,A -85,B 0,C 180,E1 -5202.167,E2 -5202.167} C_VEL
LIN {X 0,Y 516.721,Z 239.298,A -85,B 0,C 180,E1 -5205.024,E2 -5205.024} C_VEL
LIN {X 0,Y 516.716,Z 242.8,A -85,B 0,C 180,E1 -5206.199,E2 -5206.199} C_VEL
LIN {X 0,Y 518.481,Z 252.68,A -85,B 0,C 180,E1 -5206.478,E2 -5206.478} C_VEL
LIN {X 0,Y 518.285,Z 265.623,A -85,B 0,C 180,E1 -5206.922,E2 -5206.922} C_VEL
LIN {X 0,Y 517.99,Z 278.283,A -85,B 0,C 180,E1 -5207.524,E2 -5207.524} C_VEL
LIN {X 0,Y 517.76,Z 289.874,A -85,B 0,C 180,E1 -5208.252,E2 -5208.252} C_VEL
LIN {X 0,Y 517.414,Z 301.023,A -85,B 0,C 180,E1 -5209.137,E2 -5209.137} C_VEL
LIN {X 0,Y 517.161,Z 310.06,A -85,B 0,C 180,E1 -5210.022,E2 -5210.022} C_VEL
LIN {X 0,Y 516.946,Z 318.309,A -85,B 0,C 180,E1 -5211.005,E2 -5211.005} C_VEL
LIN {X 0,Y 516.686,Z 326.363,A -85,B 0,C 180,E1 -5212.182,E2 -5212.182} C_VEL
LIN {X 0,Y 516.544,Z 332.685,A -85,B 0,C 180,E1 -5213.33,E2 -5213.33} C_VEL
LIN {X 0,Y 516.405,Z 337.959,A -85,B 0,C 180,E1 -5214.533,E2 -5214.533} C_VEL
LIN {X 0,Y 516.385,Z 341.928,A -85,B 0,C 180,E1 -5215.707,E2 -5215.707} C_VEL
LIN {X 0,Y 516.363,Z 344.858,A -85,B 0,C 180,E1 -5216.879,E2 -5216.879} C_VEL
LIN {X 0,Y 516.264,Z 346.296,A -85,B 0,C 180,E1 -5217.659,E2 -5217.659} C_VEL
LIN {X 0,Y 516.176,Z 347.897,A -85,B 0,C 180,E1 -5219.22,E2 -5219.22} C_VEL
LIN {X 0,Y 516.174,Z 348.127,A -85,B 0,C 180,E1 -5220,E2 -5220} C_VEL
LIN {X 0,Y 516.194,Z 347.347,A -85,B 0,C 180,E1 -5221.56,E2 -5221.56} C_VEL
LIN {X 0,Y 516.264,Z 346.368,A -85,B 0,C 180,E1 -5222.341,E2 -5222.341} C_VEL
LIN {X 0,Y 516.363,Z 344.978,A -85,B 0,C 180,E1 -5223.121,E2 -5223.121} C_VEL
LIN {X 0,Y 516.376,Z 342.093,A -85,B 0,C 180,E1 -5224.293,E2 -5224.293} C_VEL
LIN {X 0,Y 516.405,Z 338.173,A -85,B 0,C 180,E1 -5225.467,E2 -5225.467} C_VEL
LIN {X 0,Y 516.549,Z 332.171,A -85,B 0,C 180,E1 -5226.832,E2 -5226.832} C_VEL
LIN {X 0,Y 516.723,Z 325.529,A -85,B 0,C 180,E1 -5228.014,E2 -5228.014} C_VEL
LIN {X 0,Y 516.913,Z 317.28,A -85,B 0,C 180,E1 -5229.193,E2 -5229.193} C_VEL
LIN {X 0,Y 517.137,Z 308.824,A -85,B 0,C 180,E1 -5230.176,E2 -5230.176} C_VEL
LIN {X 0,Y 517.439,Z 298.426,A -85,B 0,C 180,E1 -5231.16,E2 -5231.16} C_VEL
LIN {X 0,Y 517.764,Z 286.975,A -85,B 0,C 180,E1 -5232.025,E2 -5232.025} C_VEL
LIN {X 0,Y 518.065,Z 274.905,A -85,B 0,C 180,E1 -5232.735,E2 -5232.735} C_VEL
LIN {X 0,Y 518.338,Z 262.776,A -85,B 0,C 180,E1 -5233.277,E2 -5233.277} C_VEL
LIN {X 0,Y 518.325,Z 251.331,A -85,B 0,C 180,E1 -5233.651,E2 -5233.651} C_VEL
LIN {X 0,Y 516.596,Z 241.905,A -85,B 0,C 180,E1 -5233.924,E2 -5233.924} C_VEL
LIN {X 0,Y 516.701,Z 233.2,A -85,B 0,C 180,E1 -5237.004,E2 -5237.004} C_VEL
LIN {X 0,Y 516.815,Z 225.121,A -85,B 0,C 180,E1 -5239.875,E2 -5239.875} C_VEL
LIN {X 0,Y 516.898,Z 216.907,A -85,B 0,C 180,E1 -5242.799,E2 -5242.799} C_VEL
LIN {X 0,Y 516.976,Z 208.565,A -85,B 0,C 180,E1 -5245.787,E2 -5245.787} C_VEL
LIN {X 0,Y 517.151,Z 199.942,A -85,B 0,C 180,E1 -5248.845,E2 -5248.845} C_VEL
LIN {X 0,Y 517.251,Z 192.333,A -85,B 0,C 180,E1 -5251.541,E2 -5251.541} C_VEL
LIN {X 0,Y 517.327,Z 183.138,A -85,B 0,C 180,E1 -5254.791,E2 -5254.791} C_VEL
LIN {X 0,Y 516.886,Z 179.103,A -85,B 0,C 180,E1 -5256.261,E2 -5256.261} C_VEL
LIN {X 0,Y 516.889,Z 179.101,A -85,B 0,C 180,E1 -5259.193,E2 -5259.193} C_VEL
LIN {X 0,Y 516.911,Z 179.095,A -85,B 0,C 180,E1 -5261.776,E2 -5261.776} C_VEL
LIN {X 0,Y 516.851,Z 179.104,A -85,B 0,C 180,E1 -5263.044,E2 -5263.044} C_VEL
LIN {X 0,Y 516.183,Z 179.187,A -85,B 0,C 180,E1 -5263.695,E2 -5263.695} C_VEL
LIN {X 0,Y 513.342,Z 179.539,A -85,B 0,C 180,E1 -5264.752,E2 -5264.752} C_VEL
LIN {X 0,Y 510.941,Z 179.84,A -85,B 0,C 180,E1 -5265.603,E2 -5265.603} C_VEL
LIN {X 0,Y 509.908,Z 179.97,A -85,B 0,C 180,E1 -5266.261,E2 -5266.261} C_VEL
LIN {X 0,Y 509.822,Z 179.978,A -85,B 0,C 180,E1 -5266.483,E2 -5266.483} C_VEL
LIN {X 0,Y 509.844,Z 179.979,A -85,B 0,C 180,E1 -5269.302,E2 -5269.302} C_VEL
LIN {X 0,Y 509.821,Z 179.98,A -85,B 0,C 180,E1 -5271.791,E2 -5271.791} C_VEL
LIN {X 0,Y 509.815,Z 179.98,A -85,B 0,C 180,E1 -5274.62,E2 -5274.62} C_VEL
LIN {X 0,Y 509.865,Z 179.975,A -85,B 0,C 180,E1 -5277.48,E2 -5277.48} C_VEL
LIN {X 0,Y 509.771,Z 179.99,A -85,B 0,C 180,E1 -5280.292,E2 -5280.292} C_VEL
LIN {X 0,Y 509.661,Z 180.004,A -85,B 0,C 180,E1 -5281.142,E2 -5281.142} C_VEL
LIN {X 0,Y 509.646,Z 183.23,A -85,B 0,C 180,E1 -5283.814,E2 -5283.814} C_VEL
LIN {X 0,Y 509.565,Z 186.551,A -85,B 0,C 180,E1 -5286.423,E2 -5286.423} C_VEL
LIN {X 0,Y 509.492,Z 190.724,A -85,B 0,C 180,E1 -5289.719,E2 -5289.719} C_VEL
LIN {X 0,Y 509.419,Z 194.042,A -85,B 0,C 180,E1 -5292.33,E2 -5292.33} C_VEL
LIN {X 0,Y 509.393,Z 198.427,A -85,B 0,C 180,E1 -5295.62,E2 -5295.62} C_VEL
LIN {X 0,Y 509.394,Z 203.024,A -85,B 0,C 180,E1 -5298.862,E2 -5298.862} C_VEL
LIN {X 0,Y 509.357,Z 207.045,A -85,B 0,C 180,E1 -5301.519,E2 -5301.519} C_VEL
LIN {X 0,Y 510.709,Z 214.762,A -85,B 0,C 180,E1 -5301.84,E2 -5301.84} C_VEL
LIN {X 0,Y 510.603,Z 224.035,A -85,B 0,C 180,E1 -5302.316,E2 -5302.316} C_VEL
LIN {X 0,Y 510.521,Z 230.933,A -85,B 0,C 180,E1 -5302.796,E2 -5302.796} C_VEL
LIN {X 0,Y 510.338,Z 237.507,A -85,B 0,C 180,E1 -5303.376,E2 -5303.376} C_VEL
LIN {X 0,Y 510.287,Z 243.669,A -85,B 0,C 180,E1 -5304.07,E2 -5304.07} C_VEL
LIN {X 0,Y 510.148,Z 249.165,A -85,B 0,C 180,E1 -5304.862,E2 -5304.862} C_VEL
LIN {X 0,Y 509.947,Z 253.427,A -85,B 0,C 180,E1 -5305.652,E2 -5305.652} C_VEL
LIN {X 0,Y 509.804,Z 258.073,A -85,B 0,C 180,E1 -5306.838,E2 -5306.838} C_VEL
LIN {X 0,Y 509.633,Z 260.229,A -85,B 0,C 180,E1 -5307.628,E2 -5307.628} C_VEL
LIN {X 0,Y 509.631,Z 261.699,A -85,B 0,C 180,E1 -5308.419,E2 -5308.419} C_VEL
LIN {X 0,Y 509.575,Z 262.577,A -85,B 0,C 180,E1 -5309.209,E2 -5309.209} C_VEL
LIN {X 0,Y 509.556,Z 262.886,A -85,B 0,C 180,E1 -5309.999,E2 -5309.999} C_VEL
LIN {X 0,Y 509.569,Z 262.644,A -85,B 0,C 180,E1 -5310.789,E2 -5310.789} C_VEL
LIN {X 0,Y 509.539,Z 261.848,A -85,B 0,C 180,E1 -5311.58,E2 -5311.58} C_VEL
LIN {X 0,Y 509.74,Z 259.485,A -85,B 0,C 180,E1 -5312.765,E2 -5312.765} C_VEL
LIN {X 0,Y 509.869,Z 255.571,A -85,B 0,C 180,E1 -5313.951,E2 -5313.951} C_VEL
LIN {X 0,Y 510.1,Z 250.853,A -85,B 0,C 180,E1 -5314.939,E2 -5314.939} C_VEL
LIN {X 0,Y 510.24,Z 244.416,A -85,B 0,C 180,E1 -5315.928,E2 -5315.928} C_VEL
LIN {X 0,Y 510.341,Z 237.438,A -85,B 0,C 180,E1 -5316.721,E2 -5316.721} C_VEL
LIN {X 0,Y 510.523,Z 229.977,A -85,B 0,C 180,E1 -5317.372,E2 -5317.372} C_VEL
LIN {X 0,Y 510.629,Z 221.799,A -85,B 0,C 180,E1 -5317.91,E2 -5317.91} C_VEL
LIN {X 0,Y 510.664,Z 213.362,A -85,B 0,C 180,E1 -5318.308,E2 -5318.308} C_VEL
LIN {X 0,Y 509.367,Z 207.034,A -85,B 0,C 180,E1 -5318.579,E2 -5318.579} C_VEL
LIN {X 0,Y 509.434,Z 202.455,A -85,B 0,C 180,E1 -5321.622,E2 -5321.622} C_VEL
LIN {X 0,Y 509.393,Z 197.438,A -85,B 0,C 180,E1 -5325.196,E2 -5325.196} C_VEL
LIN {X 0,Y 509.427,Z 193.119,A -85,B 0,C 180,E1 -5328.499,E2 -5328.499} C_VEL
LIN {X 0,Y 509.461,Z 189.918,A -85,B 0,C 180,E1 -5331.017,E2 -5331.017} C_VEL
LIN {X 0,Y 509.562,Z 186.707,A -85,B 0,C 180,E1 -5333.575,E2 -5333.575} C_VEL
LIN {X 0,Y 509.643,Z 183.232,A -85,B 0,C 180,E1 -5336.317,E2 -5336.317} C_VEL
LIN {X 0,Y 509.671,Z 180.002,A -85,B 0,C 180,E1 -5338.856,E2 -5338.856} C_VEL
LIN {X 0,Y 509.814,Z 179.984,A -85,B 0,C 180,E1 -5341.589,E2 -5341.589} C_VEL
LIN {X 0,Y 509.848,Z 179.973,A -85,B 0,C 180,E1 -5344.412,E2 -5344.412} C_VEL
LIN {X 0,Y 509.813,Z 179.985,A -85,B 0,C 180,E1 -5347.339,E2 -5347.339} C_VEL
LIN {X 0,Y 509.833,Z 179.975,A -85,B 0,C 180,E1 -5350.381,E2 -5350.381} C_VEL
LIN {X 0,Y 509.834,Z 179.982,A -85,B 0,C 180,E1 -5353.063,E2 -5353.063} C_VEL
LIN {X 0,Y 509.823,Z 179.975,A -85,B 0,C 180,E1 -5355.791,E2 -5355.791} C_VEL
LIN {X 0,Y 509.852,Z 179.976,A -85,B 0,C 180,E1 -5358.574,E2 -5358.574} C_VEL
LIN {X 0,Y 509.845,Z 179.972,A -85,B 0,C 180,E1 -5361.785,E2 -5361.785} C_VEL
LIN {X 0,Y 509.839,Z 179.981,A -85,B 0,C 180,E1 -5364.622,E2 -5364.622} C_VEL
LIN {X 0,Y 509.858,Z 179.97,A -85,B 0,C 180,E1 -5367.48,E2 -5367.48} C_VEL
LIN {X 0,Y 509.873,Z 179.974,A -85,B 0,C 180,E1 -5370.268,E2 -5370.268} C_VEL
LIN {X 0,Y 509.878,Z 179.969,A -85,B 0,C 180,E1 -5372.944,E2 -5372.944} C_VEL
LIN {X 0,Y 509.86,Z 179.969,A -85,B 0,C 180,E1 -5375.573,E2 -5375.573} C_VEL
LIN {X 0,Y 509.813,Z 179.981,A -85,B 0,C 180,E1 -5378.148,E2 -5378.148} C_VEL
LIN {X 0,Y 509.855,Z 179.97,A -85,B 0,C 180,E1 -5380.681,E2 -5380.681} C_VEL
LIN {X 0,Y 509.877,Z 179.97,A -85,B 0,C 180,E1 -5383.174,E2 -5383.174} C_VEL
LIN {X 0,Y 509.854,Z 179.975,A -85,B 0,C 180,E1 -5385.634,E2 -5385.634} C_VEL
LIN {X 0,Y 509.907,Z 179.965,A -85,B 0,C 180,E1 -5388.874,E2 -5388.874} C_VEL
LIN {X 0,Y 509.941,Z 179.961,A -85,B 0,C 180,E1 -5392.078,E2 -5392.078} C_VEL
LIN {X 0,Y 509.969,Z 179.955,A -85,B 0,C 180,E1 -5394.464,E2 -5394.464} C_VEL
LIN {X 0,Y 510.04,Z 179.949,A -85,B 0,C 180,E1 -5397.631,E2 -5397.631} C_VEL
LIN {X 0,Y 510.054,Z 179.949,A -85,B 0,C 180,E1 -5400.789,E2 -5400.789} C_VEL
LIN {X 0,Y 509.94,Z 179.963,A -85,B 0,C 180,E1 -5403.16,E2 -5403.16} C_VEL
LIN {X 0,Y 509.938,Z 179.963,A -85,B 0,C 180,E1 -5406.33,E2 -5406.33} C_VEL
LIN {X 0,Y 509.898,Z 179.969,A -85,B 0,C 180,E1 -5408.72,E2 -5408.72} C_VEL
LIN {X 0,Y 509.892,Z 179.969,A -85,B 0,C 180,E1 -5411.932,E2 -5411.932} C_VEL
LIN {X 0,Y 509.882,Z 179.968,A -85,B 0,C 180,E1 -5415.242,E2 -5415.242} C_VEL
LIN {X 0,Y 509.844,Z 179.977,A -85,B 0,C 180,E1 -5418.484,E2 -5418.484} C_VEL
LIN {X 0,Y 509.832,Z 179.975,A -85,B 0,C 180,E1 -5421.003,E2 -5421.003} C_VEL
LIN {X 0,Y 509.805,Z 179.982,A -85,B 0,C 180,E1 -5423.565,E2 -5423.565} C_VEL
LIN {X 0,Y 509.802,Z 179.98,A -85,B 0,C 180,E1 -5426.357,E2 -5426.357} C_VEL
LIN {X 0,Y 509.821,Z 179.977,A -85,B 0,C 180,E1 -5428.848,E2 -5428.848} C_VEL
LIN {X 0,Y 509.807,Z 179.985,A -85,B 0,C 180,E1 -5431.591,E2 -5431.591} C_VEL
LIN {X 0,Y 509.828,Z 179.973,A -85,B 0,C 180,E1 -5434.415,E2 -5434.415} C_VEL
LIN {X 0,Y 509.797,Z 179.985,A -85,B 0,C 180,E1 -5437.343,E2 -5437.343} C_VEL
LIN {X 0,Y 509.808,Z 179.975,A -85,B 0,C 180,E1 -5440.385,E2 -5440.385} C_VEL
LIN {X 0,Y 509.796,Z 179.986,A -85,B 0,C 180,E1 -5443.061,E2 -5443.061} C_VEL
LIN {X 0,Y 509.814,Z 179.977,A -85,B 0,C 180,E1 -5445.794,E2 -5445.794} C_VEL
LIN {X 0,Y 509.848,Z 179.974,A -85,B 0,C 180,E1 -5448.576,E2 -5448.576} C_VEL
LIN {X 0,Y 509.845,Z 179.975,A -85,B 0,C 180,E1 -5451.788,E2 -5451.788} C_VEL
LIN {X 0,Y 509.825,Z 179.979,A -85,B 0,C 180,E1 -5454.623,E2 -5454.623} C_VEL
LIN {X 0,Y 509.847,Z 180.007,A -85,B 0,C 180,E1 -5457.301,E2 -5457.301} C_VEL
LIN {X 0,Y 512.54,Z 191.824,A -85,B 0,C 180,E1 -5459.753,E2 -5459.753} C_VEL
LIN {X 0,Y 513.127,Z 195.562,A -85,B 0,C 180,E1 -5460.459,E2 -5460.459} C_VEL
LIN {X 0,Y 512.313,Z 212.223,A -85,B 0,C 180,E1 -5463.305,E2 -5463.305} C_VEL
LIN {X 0,Y 511.549,Z 232.014,A -85,B 0,C 180,E1 -5466.522,E2 -5466.522} C_VEL
LIN {X 0,Y 510.955,Z 251.234,A -85,B 0,C 180,E1 -5469.572,E2 -5469.572} C_VEL
LIN {X 0,Y 510.431,Z 268.973,A -85,B 0,C 180,E1 -5472.369,E2 -5472.369} C_VEL
LIN {X 0,Y 510.013,Z 289.699,A -85,B 0,C 180,E1 -5475.64,E2 -5475.64} C_VEL
LIN {X 0,Y 509.913,Z 292.196,A -85,B 0,C 180,E1 -5476.044,E2 -5476.044} C_VEL
LIN {X 0,Y 511.139,Z 307.147,A -85,B 0,C 180,E1 -5476.408,E2 -5476.408} C_VEL
LIN {X 0,Y 510.915,Z 319.487,A -85,B 0,C 180,E1 -5476.832,E2 -5476.832} C_VEL
LIN {X 0,Y 510.6,Z 331.458,A -85,B 0,C 180,E1 -5477.38,E2 -5477.38} C_VEL
LIN {X 0,Y 510.388,Z 343.242,A -85,B 0,C 180,E1 -5478.081,E2 -5478.081} C_VEL
LIN {X 0,Y 510.104,Z 353.803,A -85,B 0,C 180,E1 -5478.88,E2 -5478.88} C_VEL
LIN {X 0,Y 509.874,Z 364.403,A -85,B 0,C 180,E1 -5479.879,E2 -5479.879} C_VEL
LIN {X 0,Y 509.677,Z 373.014,A -85,B 0,C 180,E1 -5480.877,E2 -5480.877} C_VEL
LIN {X 0,Y 509.52,Z 381.396,A -85,B 0,C 180,E1 -5482.073,E2 -5482.073} C_VEL
LIN {X 0,Y 509.389,Z 388.741,A -85,B 0,C 180,E1 -5483.404,E2 -5483.404} C_VEL
LIN {X 0,Y 509.365,Z 394.91,A -85,B 0,C 180,E1 -5484.856,E2 -5484.856} C_VEL
LIN {X 0,Y 509.396,Z 398.748,A -85,B 0,C 180,E1 -5486.045,E2 -5486.045} C_VEL
LIN {X 0,Y 509.325,Z 400.696,A -85,B 0,C 180,E1 -5486.837,E2 -5486.837} C_VEL
LIN {X 0,Y 509.287,Z 402.178,A -85,B 0,C 180,E1 -5487.628,E2 -5487.628} C_VEL
LIN {X 0,Y 509.246,Z 403.234,A -85,B 0,C 180,E1 -5488.419,E2 -5488.419} C_VEL
LIN {X 0,Y 509.269,Z 403.881,A -85,B 0,C 180,E1 -5489.21,E2 -5489.21} C_VEL
LIN {X 0,Y 509.282,Z 404.107,A -85,B 0,C 180,E1 -5490.001,E2 -5490.001} C_VEL
LIN {X 0,Y 509.252,Z 403.19,A -85,B 0,C 180,E1 -5491.583,E2 -5491.583} C_VEL
LIN {X 0,Y 509.286,Z 402.186,A -85,B 0,C 180,E1 -5492.374,E2 -5492.374} C_VEL
LIN {X 0,Y 509.328,Z 400.66,A -85,B 0,C 180,E1 -5493.165,E2 -5493.165} C_VEL
LIN {X 0,Y 509.387,Z 397.576,A -85,B 0,C 180,E1 -5494.353,E2 -5494.353} C_VEL
LIN {X 0,Y 509.398,Z 391.68,A -85,B 0,C 180,E1 -5495.94,E2 -5495.94} C_VEL
LIN {X 0,Y 509.455,Z 385.816,A -85,B 0,C 180,E1 -5497.133,E2 -5497.133} C_VEL
LIN {X 0,Y 509.578,Z 378.471,A -85,B 0,C 180,E1 -5498.327,E2 -5498.327} C_VEL
LIN {X 0,Y 509.737,Z 369.351,A -85,B 0,C 180,E1 -5499.524,E2 -5499.524} C_VEL
LIN {X 0,Y 509.946,Z 359.943,A -85,B 0,C 180,E1 -5500.523,E2 -5500.523} C_VEL
LIN {X 0,Y 510.247,Z 348.192,A -85,B 0,C 180,E1 -5501.521,E2 -5501.521} C_VEL
LIN {X 0,Y 510.519,Z 336.692,A -85,B 0,C 180,E1 -5502.302,E2 -5502.302} C_VEL
LIN {X 0,Y 510.797,Z 325.133,A -85,B 0,C 180,E1 -5502.92,E2 -5502.92} C_VEL
LIN {X 0,Y 511.035,Z 311.948,A -85,B 0,C 180,E1 -5503.445,E2 -5503.445} C_VEL
LIN {X 0,Y 511.04,Z 303.812,A -85,B 0,C 180,E1 -5503.686,E2 -5503.686} C_VEL
LIN {X 0,Y 509.92,Z 292.211,A -85,B 0,C 180,E1 -5503.958,E2 -5503.958} C_VEL
LIN {X 0,Y 510.372,Z 271.514,A -85,B 0,C 180,E1 -5507.222,E2 -5507.222} C_VEL
LIN {X 0,Y 510.961,Z 251.251,A -85,B 0,C 180,E1 -5510.43,E2 -5510.43} C_VEL
LIN {X 0,Y 511.607,Z 230.678,A -85,B 0,C 180,E1 -5513.692,E2 -5513.692} C_VEL
LIN {X 0,Y 512.319,Z 212.181,A -85,B 0,C 180,E1 -5516.697,E2 -5516.697} C_VEL
LIN {X 0,Y 513.117,Z 195.497,A -85,B 0,C 180,E1 -5519.544,E2 -5519.544} C_VEL
LIN {X 0,Y 511.751,Z 188.101,A -85,B 0,C 180,E1 -5520.998,E2 -5520.998} C_VEL
LIN {X 0,Y 509.828,Z 179.984,A -85,B 0,C 180,E1 -5522.695,E2 -5522.695} C_VEL
LIN {X 0,Y 509.824,Z 179.982,A -85,B 0,C 180,E1 -5525.578,E2 -5525.578} C_VEL
LIN {X 0,Y 509.852,Z 179.979,A -85,B 0,C 180,E1 -5528.339,E2 -5528.339} C_VEL
LIN {X 0,Y 509.86,Z 179.973,A -85,B 0,C 180,E1 -5531.426,E2 -5531.426} C_VEL
LIN {X 0,Y 509.844,Z 179.976,A -85,B 0,C 180,E1 -5534.67,E2 -5534.67} C_VEL
LIN {X 0,Y 509.86,Z 179.974,A -85,B 0,C 180,E1 -5538.104,E2 -5538.104} C_VEL
LIN {X 0,Y 509.838,Z 179.981,A -85,B 0,C 180,E1 -5540.647,E2 -5540.647} C_VEL
LIN {X 0,Y 509.794,Z 179.984,A -85,B 0,C 180,E1 -5543.644,E2 -5543.644} C_VEL
LIN {X 0,Y 509.812,Z 180.058,A -85,B 0,C 180,E1 -5545.404,E2 -5545.404} C_VEL
LIN {X 0,Y 510.038,Z 186.245,A -85,B 0,C 180,E1 -5547.198,E2 -5547.198} C_VEL
LIN {X 0,Y 509.963,Z 194.931,A -85,B 0,C 180,E1 -5549.8,E2 -5549.8} C_VEL
LIN {X 0,Y 509.954,Z 203.522,A -85,B 0,C 180,E1 -5552.504,E2 -5552.504} C_VEL
LIN {X 0,Y 509.938,Z 211.419,A -85,B 0,C 180,E1 -5555.125,E2 -5555.125} C_VEL
LIN {X 0,Y 509.902,Z 219.465,A -85,B 0,C 180,E1 -5557.794,E2 -5557.794} C_VEL
LIN {X 0,Y 509.835,Z 227.873,A -85,B 0,C 180,E1 -5560.68,E2 -5560.68} C_VEL
LIN {X 0,Y 509.711,Z 236.181,A -85,B 0,C 180,E1 -5563.581,E2 -5563.581} C_VEL
LIN {X 0,Y 509.675,Z 243.21,A -85,B 0,C 180,E1 -5566.011,E2 -5566.011} C_VEL
LIN {X 0,Y 511.597,Z 253.653,A -85,B 0,C 180,E1 -5566.318,E2 -5566.318} C_VEL
LIN {X 0,Y 511.339,Z 266.939,A -85,B 0,C 180,E1 -5566.791,E2 -5566.791} C_VEL
LIN {X 0,Y 511.007,Z 279.86,A -85,B 0,C 180,E1 -5567.43,E2 -5567.43} C_VEL
LIN {X 0,Y 510.798,Z 291.459,A -85,B 0,C 180,E1 -5568.19,E2 -5568.19} C_VEL
LIN {X 0,Y 510.414,Z 302.399,A -85,B 0,C 180,E1 -5569.086,E2 -5569.086} C_VEL
LIN {X 0,Y 510.108,Z 312.126,A -85,B 0,C 180,E1 -5570.083,E2 -5570.083} C_VEL
LIN {X 0,Y 509.852,Z 321.529,A -85,B 0,C 180,E1 -5571.279,E2 -5571.279} C_VEL
LIN {X 0,Y 509.6,Z 329.033,A -85,B 0,C 180,E1 -5572.472,E2 -5572.472} C_VEL
LIN {X 0,Y 509.488,Z 335.032,A -85,B 0,C 180,E1 -5573.664,E2 -5573.664} C_VEL
LIN {X 0,Y 509.278,Z 339.78,A -85,B 0,C 180,E1 -5574.854,E2 -5574.854} C_VEL
LIN {X 0,Y 509.309,Z 343.396,A -85,B 0,C 180,E1 -5576.044,E2 -5576.044} C_VEL
LIN {X 0,Y 509.304,Z 345.247,A -85,B 0,C 180,E1 -5576.836,E2 -5576.836} C_VEL
LIN {X 0,Y 509.196,Z 346.685,A -85,B 0,C 180,E1 -5577.627,E2 -5577.627} C_VEL
LIN {X 0,Y 509.089,Z 348.286,A -85,B 0,C 180,E1 -5579.209,E2 -5579.209} C_VEL
LIN {X 0,Y 509.086,Z 348.513,A -85,B 0,C 180,E1 -5580,E2 -5580} C_VEL
LIN {X 0,Y 509.087,Z 348.317,A -85,B 0,C 180,E1 -5580.791,E2 -5580.791} C_VEL
LIN {X 0,Y 509.196,Z 346.735,A -85,B 0,C 180,E1 -5582.373,E2 -5582.373} C_VEL
LIN {X 0,Y 509.304,Z 345.34,A -85,B 0,C 180,E1 -5583.164,E2 -5583.164} C_VEL
LIN {X 0,Y 509.305,Z 342.441,A -85,B 0,C 180,E1 -5584.353,E2 -5584.353} C_VEL
LIN {X 0,Y 509.35,Z 338.503,A -85,B 0,C 180,E1 -5585.543,E2 -5585.543} C_VEL
LIN {X 0,Y 509.489,Z 332.683,A -85,B 0,C 180,E1 -5586.885,E2 -5586.885} C_VEL
LIN {X 0,Y 509.677,Z 325.807,A -85,B 0,C 180,E1 -5588.125,E2 -5588.125} C_VEL
LIN {X 0,Y 509.909,Z 317.535,A -85,B 0,C 180,E1 -5589.32,E2 -5589.32} C_VEL
LIN {X 0,Y 510.142,Z 309.039,A -85,B 0,C 180,E1 -5590.317,E2 -5590.317} C_VEL
LIN {X 0,Y 510.484,Z 298.617,A -85,B 0,C 180,E1 -5591.314,E2 -5591.314} C_VEL
LIN {X 0,Y 510.796,Z 287.118,A -85,B 0,C 180,E1 -5592.191,E2 -5592.191} C_VEL
LIN {X 0,Y 511.136,Z 275.022,A -85,B 0,C 180,E1 -5592.911,E2 -5592.911} C_VEL
LIN {X 0,Y 511.44,Z 262.84,A -85,B 0,C 180,E1 -5593.459,E2 -5593.459} C_VEL
LIN {X 0,Y 511.387,Z 252.046,A -85,B 0,C 180,E1 -5593.821,E2 -5593.821} C_VEL
LIN {X 0,Y 509.533,Z 242.181,A -85,B 0,C 180,E1 -5594.121,E2 -5594.121} C_VEL
LIN {X 0,Y 509.652,Z 234.564,A -85,B 0,C 180,E1 -5596.833,E2 -5596.833} C_VEL
LIN {X 0,Y 509.765,Z 226.432,A -85,B 0,C 180,E1 -5599.742,E2 -5599.742} C_VEL
LIN {X 0,Y 509.862,Z 218.172,A -85,B 0,C 180,E1 -5602.703,E2 -5602.703} C_VEL
LIN {X 0,Y 509.971,Z 210.956,A -85,B 0,C 180,E1 -5605.291,E2 -5605.291} C_VEL
LIN {X 0,Y 510.103,Z 202.978,A -85,B 0,C 180,E1 -5608.143,E2 -5608.143} C_VEL
LIN {X 0,Y 510.162,Z 195.969,A -85,B 0,C 180,E1 -5610.645,E2 -5610.645} C_VEL
LIN {X 0,Y 510.274,Z 188.131,A -85,B 0,C 180,E1 -5613.43,E2 -5613.43} C_VEL
LIN {X 0,Y 510.218,Z 182.748,A -85,B 0,C 180,E1 -5615.347,E2 -5615.347} C_VEL
LIN {X 0,Y 509.844,Z 179.98,A -85,B 0,C 180,E1 -5616.403,E2 -5616.403} C_VEL
LIN {X 0,Y 509.838,Z 179.981,A -85,B 0,C 180,E1 -5619.47,E2 -5619.47} C_VEL
LIN {X 0,Y 509.818,Z 179.982,A -85,B 0,C 180,E1 -5622.492,E2 -5622.492} C_VEL
LIN {X 0,Y 509.844,Z 179.974,A -85,B 0,C 180,E1 -5625.33,E2 -5625.33} C_VEL
LIN {X 0,Y 509.822,Z 179.978,A -85,B 0,C 180,E1 -5626.483,E2 -5626.483} C_VEL
LIN {X 0,Y 509.148,Z 180.065,A -85,B 0,C 180,E1 -5627.142,E2 -5627.142} C_VEL
LIN {X 0,Y 506.285,Z 180.419,A -85,B 0,C 180,E1 -5628.212,E2 -5628.212} C_VEL
LIN {X 0,Y 503.88,Z 180.723,A -85,B 0,C 180,E1 -5629.074,E2 -5629.074} C_VEL
LIN {X 0,Y 502.865,Z 180.845,A -85,B 0,C 180,E1 -5629.74,E2 -5629.74} C_VEL
LIN {X 0,Y 502.792,Z 180.854,A -85,B 0,C 180,E1 -5629.965,E2 -5629.965} C_VEL
LIN {X 0,Y 502.725,Z 180.864,A -85,B 0,C 180,E1 -5633.048,E2 -5633.048} C_VEL
LIN {X 0,Y 502.791,Z 180.856,A -85,B 0,C 180,E1 -5636.004,E2 -5636.004} C_VEL
LIN {X 0,Y 502.792,Z 180.859,A -85,B 0,C 180,E1 -5638.856,E2 -5638.856} C_VEL
LIN {X 0,Y 502.659,Z 180.876,A -85,B 0,C 180,E1 -5640.701,E2 -5640.701} C_VEL
LIN {X 0,Y 502.584,Z 181.415,A -85,B 0,C 180,E1 -5641.761,E2 -5641.761} C_VEL
LIN {X 0,Y 502.571,Z 184.65,A -85,B 0,C 180,E1 -5644.309,E2 -5644.309} C_VEL
LIN {X 0,Y 502.48,Z 188.555,A -85,B 0,C 180,E1 -5647.387,E2 -5647.387} C_VEL
LIN {X 0,Y 502.389,Z 192.332,A -85,B 0,C 180,E1 -5650.382,E2 -5650.382} C_VEL
LIN {X 0,Y 502.32,Z 195.588,A -85,B 0,C 180,E1 -5652.913,E2 -5652.913} C_VEL
LIN {X 0,Y 502.363,Z 198.909,A -85,B 0,C 180,E1 -5655.414,E2 -5655.414} C_VEL
LIN {X 0,Y 502.344,Z 203.557,A -85,B 0,C 180,E1 -5658.704,E2 -5658.704} C_VEL
LIN {X 0,Y 502.32,Z 207.573,A -85,B 0,C 180,E1 -5661.349,E2 -5661.349} C_VEL
LIN {X 0,Y 503.81,Z 215.466,A -85,B 0,C 180,E1 -5661.678,E2 -5661.678} C_VEL
LIN {X 0,Y 503.743,Z 223.519,A -85,B 0,C 180,E1 -5662.074,E2 -5662.074} C_VEL
LIN {X 0,Y 503.607,Z 231.744,A -85,B 0,C 180,E1 -5662.639,E2 -5662.639} C_VEL
LIN {X 0,Y 503.422,Z 238.943,A -85,B 0,C 180,E1 -5663.285,E2 -5663.285} C_VEL
LIN {X 0,Y 503.362,Z 245.026,A -85,B 0,C 180,E1 -5663.988,E2 -5663.988} C_VEL
LIN {X 0,Y 503.194,Z 250.417,A -85,B 0,C 180,E1 -5664.79,E2 -5664.79} C_VEL
LIN {X 0,Y 502.966,Z 254.613,A -85,B 0,C 180,E1 -5665.591,E2 -5665.591} C_VEL
LIN {X 0,Y 502.809,Z 259.172,A -85,B 0,C 180,E1 -5666.794,E2 -5666.794} C_VEL
LIN {X 0,Y 502.624,Z 261.279,A -85,B 0,C 180,E1 -5667.595,E2 -5667.595} C_VEL
LIN {X 0,Y 502.622,Z 262.71,A -85,B 0,C 180,E1 -5668.396,E2 -5668.396} C_VEL
LIN {X 0,Y 502.56,Z 263.561,A -85,B 0,C 180,E1 -5669.198,E2 -5669.198} C_VEL
LIN {X 0,Y 502.538,Z 263.859,A -85,B 0,C 180,E1 -5669.999,E2 -5669.999} C_VEL
LIN {X 0,Y 502.553,Z 263.624,A -85,B 0,C 180,E1 -5670.8,E2 -5670.8} C_VEL
LIN {X 0,Y 502.539,Z 262.85,A -85,B 0,C 180,E1 -5671.602,E2 -5671.602} C_VEL
LIN {X 0,Y 502.739,Z 260.549,A -85,B 0,C 180,E1 -5672.803,E2 -5672.803} C_VEL
LIN {X 0,Y 502.902,Z 256.717,A -85,B 0,C 180,E1 -5674.006,E2 -5674.006} C_VEL
LIN {X 0,Y 503.141,Z 252.076,A -85,B 0,C 180,E1 -5675.007,E2 -5675.007} C_VEL
LIN {X 0,Y 503.293,Z 245.738,A -85,B 0,C 180,E1 -5676.011,E2 -5676.011} C_VEL
LIN {X 0,Y 503.409,Z 238.863,A -85,B 0,C 180,E1 -5676.814,E2 -5676.814} C_VEL
LIN {X 0,Y 503.625,Z 232.351,A -85,B 0,C 180,E1 -5677.402,E2 -5677.402} C_VEL
LIN {X 0,Y 503.683,Z 224.632,A -85,B 0,C 180,E1 -5677.95,E2 -5677.95} C_VEL
LIN {X 0,Y 503.836,Z 215.241,A -85,B 0,C 180,E1 -5678.421,E2 -5678.421} C_VEL
LIN {X 0,Y 502.286,Z 207.564,A -85,B 0,C 180,E1 -5678.751,E2 -5678.751} C_VEL
LIN {X 0,Y 502.377,Z 203.127,A -85,B 0,C 180,E1 -5681.687,E2 -5681.687} C_VEL
LIN {X 0,Y 502.336,Z 197.908,A -85,B 0,C 180,E1 -5685.415,E2 -5685.415} C_VEL
LIN {X 0,Y 502.362,Z 193.545,A -85,B 0,C 180,E1 -5688.769,E2 -5688.769} C_VEL
LIN {X 0,Y 502.423,Z 190.315,A -85,B 0,C 180,E1 -5691.326,E2 -5691.326} C_VEL
LIN {X 0,Y 502.506,Z 187.05,A -85,B 0,C 180,E1 -5693.927,E2 -5693.927} C_VEL
LIN {X 0,Y 502.591,Z 183.695,A -85,B 0,C 180,E1 -5696.58,E2 -5696.58} C_VEL
LIN {X 0,Y 502.607,Z 181.372,A -85,B 0,C 180,E1 -5698.386,E2 -5698.386} C_VEL
LIN {X 0,Y 502.735,Z 180.865,A -85,B 0,C 180,E1 -5699.919,E2 -5699.919} C_VEL
LIN {X 0,Y 502.828,Z 180.849,A -85,B 0,C 180,E1 -5703.03,E2 -5703.03} C_VEL
LIN {X 0,Y 502.776,Z 180.856,A -85,B 0,C 180,E1 -5705.949,E2 -5705.949} C_VEL
LIN {X 0,Y 502.796,Z 180.855,A -85,B 0,C 180,E1 -5708.975,E2 -5708.975} C_VEL
LIN {X 0,Y 502.824,Z 180.847,A -85,B 0,C 180,E1 -5712.135,E2 -5712.135} C_VEL
LIN {X 0,Y 502.794,Z 180.853,A -85,B 0,C 180,E1 -5715.467,E2 -5715.467} C_VEL
LIN {X 0,Y 502.813,Z 180.854,A -85,B 0,C 180,E1 -5718.933,E2 -5718.933} C_VEL
LIN {X 0,Y 502.788,Z 180.852,A -85,B 0,C 180,E1 -5722.045,E2 -5722.045} C_VEL
LIN {X 0,Y 502.802,Z 180.852,A -85,B 0,C 180,E1 -5725.034,E2 -5725.034} C_VEL
LIN {X 0,Y 502.78,Z 180.854,A -85,B 0,C 180,E1 -5727.915,E2 -5727.915} C_VEL
LIN {X 0,Y 502.83,Z 180.848,A -85,B 0,C 180,E1 -5730.712,E2 -5730.712} C_VEL
LIN {X 0,Y 502.871,Z 180.842,A -85,B 0,C 180,E1 -5733.434,E2 -5733.434} C_VEL
LIN {X 0,Y 502.782,Z 180.858,A -85,B 0,C 180,E1 -5736.086,E2 -5736.086} C_VEL
LIN {X 0,Y 502.774,Z 180.852,A -85,B 0,C 180,E1 -5738.688,E2 -5738.688} C_VEL
LIN {X 0,Y 502.82,Z 180.848,A -85,B 0,C 180,E1 -5741.248,E2 -5741.248} C_VEL
LIN {X 0,Y 502.814,Z 180.852,A -85,B 0,C 180,E1 -5743.767,E2 -5743.767} C_VEL
LIN {X 0,Y 502.821,Z 180.848,A -85,B 0,C 180,E1 -5746.254,E2 -5746.254} C_VEL
LIN {X 0,Y 502.87,Z 180.841,A -85,B 0,C 180,E1 -5748.717,E2 -5748.717} C_VEL
LIN {X 0,Y 502.891,Z 180.839,A -85,B 0,C 180,E1 -5751.966,E2 -5751.966} C_VEL
LIN {X 0,Y 502.923,Z 180.833,A -85,B 0,C 180,E1 -5754.386,E2 -5754.386} C_VEL
LIN {X 0,Y 503.01,Z 180.825,A -85,B 0,C 180,E1 -5757.598,E2 -5757.598} C_VEL
LIN {X 0,Y 503.011,Z 180.819,A -85,B 0,C 180,E1 -5760,E2 -5760} C_VEL
LIN {X 0,Y 503.01,Z 180.826,A -85,B 0,C 180,E1 -5762.402,E2 -5762.402} C_VEL
LIN {X 0,Y 502.918,Z 180.834,A -85,B 0,C 180,E1 -5765.614,E2 -5765.614} C_VEL
LIN {X 0,Y 502.888,Z 180.841,A -85,B 0,C 180,E1 -5768.034,E2 -5768.034} C_VEL
LIN {X 0,Y 502.863,Z 180.843,A -85,B 0,C 180,E1 -5771.283,E2 -5771.283} C_VEL
LIN {X 0,Y 502.831,Z 180.851,A -85,B 0,C 180,E1 -5774.571,E2 -5774.571} C_VEL
LIN {X 0,Y 502.804,Z 180.853,A -85,B 0,C 180,E1 -5777.909,E2 -5777.909} C_VEL
LIN {X 0,Y 502.817,Z 180.851,A -85,B 0,C 180,E1 -5780.537,E2 -5780.537} C_VEL
LIN {X 0,Y 502.774,Z 180.854,A -85,B 0,C 180,E1 -5783.041,E2 -5783.041} C_VEL
LIN {X 0,Y 502.764,Z 180.862,A -85,B 0,C 180,E1 -5785.68,E2 -5785.68} C_VEL
LIN {X 0,Y 502.757,Z 180.857,A -85,B 0,C 180,E1 -5788.378,E2 -5788.378} C_VEL
LIN {X 0,Y 502.78,Z 180.856,A -85,B 0,C 180,E1 -5791.144,E2 -5791.144} C_VEL
LIN {X 0,Y 502.782,Z 180.852,A -85,B 0,C 180,E1 -5793.996,E2 -5793.996} C_VEL
LIN {X 0,Y 502.754,Z 180.862,A -85,B 0,C 180,E1 -5797.177,E2 -5797.177} C_VEL
LIN {X 0,Y 502.763,Z 180.853,A -85,B 0,C 180,E1 -5800.018,E2 -5800.018} C_VEL
LIN {X 0,Y 502.795,Z 180.852,A -85,B 0,C 180,E1 -5802.2,E2 -5802.2} C_VEL
LIN {X 0,Y 502.778,Z 180.856,A -85,B 0,C 180,E1 -5805.471,E2 -5805.471} C_VEL
LIN {X 0,Y 502.813,Z 180.856,A -85,B 0,C 180,E1 -5808.935,E2 -5808.935} C_VEL
LIN {X 0,Y 502.787,Z 180.856,A -85,B 0,C 180,E1 -5812.047,E2 -5812.047} C_VEL
LIN {X 0,Y 502.794,Z 180.852,A -85,B 0,C 180,E1 -5815.035,E2 -5815.035} C_VEL
LIN {X 0,Y 502.829,Z 180.989,A -85,B 0,C 180,E1 -5816.994,E2 -5816.994} C_VEL
LIN {X 0,Y 505.751,Z 193.719,A -85,B 0,C 180,E1 -5819.677,E2 -5819.677} C_VEL
LIN {X 0,Y 506.241,Z 197.928,A -85,B 0,C 180,E1 -5820.474,E2 -5820.474} C_VEL
LIN {X 0,Y 505.429,Z 213.554,A -85,B 0,C 180,E1 -5823.189,E2 -5823.189} C_VEL
LIN {X 0,Y 504.612,Z 232.801,A -85,B 0,C 180,E1 -5826.372,E2 -5826.372} C_VEL
LIN {X 0,Y 503.98,Z 251.235,A -85,B 0,C 180,E1 -5829.35,E2 -5829.35} C_VEL
LIN {X 0,Y 503.445,Z 268.468,A -85,B 0,C 180,E1 -5832.116,E2 -5832.116} C_VEL
LIN {X 0,Y 502.92,Z 290.219,A -85,B 0,C 180,E1 -5835.639,E2 -5835.639} C_VEL
LIN {X 0,Y 502.861,Z 291.966,A -85,B 0,C 180,E1 -5835.909,E2 -5835.909} C_VEL
LIN {X 0,Y 504.142,Z 305.85,A -85,B 0,C 180,E1 -5836.228,E2 -5836.228} C_VEL
LIN {X 0,Y 503.964,Z 318.832,A -85,B 0,C 180,E1 -5836.647,E2 -5836.647} C_VEL
LIN {X 0,Y 503.613,Z 332.217,A -85,B 0,C 180,E1 -5837.268,E2 -5837.268} C_VEL
LIN {X 0,Y 503.345,Z 344.192,A -85,B 0,C 180,E1 -5838.014,E2 -5838.014} C_VEL
LIN {X 0,Y 503.018,Z 355.656,A -85,B 0,C 180,E1 -5838.925,E2 -5838.925} C_VEL
LIN {X 0,Y 502.792,Z 365.838,A -85,B 0,C 180,E1 -5839.939,E2 -5839.939} C_VEL
LIN {X 0,Y 502.607,Z 374.12,A -85,B 0,C 180,E1 -5840.95,E2 -5840.95} C_VEL
LIN {X 0,Y 502.417,Z 382.184,A -85,B 0,C 180,E1 -5842.162,E2 -5842.162} C_VEL
LIN {X 0,Y 502.303,Z 388.843,A -85,B 0,C 180,E1 -5843.415,E2 -5843.415} C_VEL
LIN {X 0,Y 502.283,Z 394.491,A -85,B 0,C 180,E1 -5844.783,E2 -5844.783} C_VEL
LIN {X 0,Y 502.325,Z 398.235,A -85,B 0,C 180,E1 -5845.99,E2 -5845.99} C_VEL
LIN {X 0,Y 502.24,Z 400.143,A -85,B 0,C 180,E1 -5846.792,E2 -5846.792} C_VEL
LIN {X 0,Y 502.214,Z 401.583,A -85,B 0,C 180,E1 -5847.595,E2 -5847.595} C_VEL
LIN {X 0,Y 502.171,Z 402.606,A -85,B 0,C 180,E1 -5848.397,E2 -5848.397} C_VEL
LIN {X 0,Y 502.197,Z 403.225,A -85,B 0,C 180,E1 -5849.199,E2 -5849.199} C_VEL
LIN {X 0,Y 502.214,Z 403.432,A -85,B 0,C 180,E1 -5850.001,E2 -5850.001} C_VEL
LIN {X 0,Y 502.181,Z 402.508,A -85,B 0,C 180,E1 -5851.605,E2 -5851.605} C_VEL
LIN {X 0,Y 502.213,Z 401.508,A -85,B 0,C 180,E1 -5852.407,E2 -5852.407} C_VEL
LIN {X 0,Y 502.273,Z 400.003,A -85,B 0,C 180,E1 -5853.209,E2 -5853.209} C_VEL
LIN {X 0,Y 502.313,Z 396.945,A -85,B 0,C 180,E1 -5854.414,E2 -5854.414} C_VEL
LIN {X 0,Y 502.305,Z 392.774,A -85,B 0,C 180,E1 -5855.622,E2 -5855.622} C_VEL
LIN {X 0,Y 502.36,Z 387.563,A -85,B 0,C 180,E1 -5856.79,E2 -5856.79} C_VEL
LIN {X 0,Y 502.448,Z 380.529,A -85,B 0,C 180,E1 -5858.042,E2 -5858.042} C_VEL
LIN {X 0,Y 502.619,Z 373.604,A -85,B 0,C 180,E1 -5859.052,E2 -5859.052} C_VEL
LIN {X 0,Y 502.794,Z 365.259,A -85,B 0,C 180,E1 -5860.064,E2 -5860.064} C_VEL
LIN {X 0,Y 503.024,Z 354.966,A -85,B 0,C 180,E1 -5861.077,E2 -5861.077} C_VEL
LIN {X 0,Y 503.269,Z 343.777,A -85,B 0,C 180,E1 -5861.959,E2 -5861.959} C_VEL
LIN {X 0,Y 503.603,Z 331.884,A -85,B 0,C 180,E1 -5862.698,E2 -5862.698} C_VEL
LIN {X 0,Y 503.903,Z 318.925,A -85,B 0,C 180,E1 -5863.306,E2 -5863.306} C_VEL
LIN {X 0,Y 504.068,Z 304.706,A -85,B 0,C 180,E1 -5863.789,E2 -5863.789} C_VEL
LIN {X 0,Y 502.931,Z 292.691,A -85,B 0,C 180,E1 -5864.079,E2 -5864.079} C_VEL
LIN {X 0,Y 502.866,Z 291.776,A -85,B 0,C 180,E1 -5864.106,E2 -5864.106} C_VEL
LIN {X 0,Y 503.379,Z 271.035,A -85,B 0,C 180,E1 -5867.469,E2 -5867.469} C_VEL
LIN {X 0,Y 504.16,Z 247.516,A -85,B 0,C 180,E1 -5871.251,E2 -5871.251} C_VEL
LIN {X 0,Y 504.727,Z 228.955,A -85,B 0,C 180,E1 -5874.254,E2 -5874.254} C_VEL
LIN {X 0,Y 505.547,Z 210.61,A -85,B 0,C 180,E1 -5877.308,E2 -5877.308} C_VEL
LIN {X 0,Y 506.264,Z 197.856,A -85,B 0,C 180,E1 -5879.527,E2 -5879.527} C_VEL
LIN {X 0,Y 505.715,Z 193.7,A -85,B 0,C 180,E1 -5880.326,E2 -5880.326} C_VEL
LIN {X 0,Y 503.053,Z 182.098,A -85,B 0,C 180,E1 -5882.761,E2 -5882.761} C_VEL
LIN {X 0,Y 502.803,Z 180.86,A -85,B 0,C 180,E1 -5883.034,E2 -5883.034} C_VEL
LIN {X 0,Y 502.771,Z 180.86,A -85,B 0,C 180,E1 -5885.952,E2 -5885.952} C_VEL
LIN {X 0,Y 502.799,Z 180.855,A -85,B 0,C 180,E1 -5888.977,E2 -5888.977} C_VEL
LIN {X 0,Y 502.825,Z 180.849,A -85,B 0,C 180,E1 -5891.066,E2 -5891.066} C_VEL
LIN {X 0,Y 502.791,Z 180.855,A -85,B 0,C 180,E1 -5894.53,E2 -5894.53} C_VEL
LIN {X 0,Y 502.8,Z 180.855,A -85,B 0,C 180,E1 -5897.861,E2 -5897.861} C_VEL
LIN {X 0,Y 502.784,Z 180.857,A -85,B 0,C 180,E1 -5900.247,E2 -5900.247} C_VEL
LIN {X 0,Y 502.755,Z 180.863,A -85,B 0,C 180,E1 -5903.051,E2 -5903.051} C_VEL
LIN {X 0,Y 502.805,Z 181.049,A -85,B 0,C 180,E1 -5905.251,E2 -5905.251} C_VEL
LIN {X 0,Y 503.103,Z 186.794,A -85,B 0,C 180,E1 -5906.947,E2 -5906.947} C_VEL
LIN {X 0,Y 502.976,Z 196.243,A -85,B 0,C 180,E1 -5909.8,E2 -5909.8} C_VEL
LIN {X 0,Y 502.961,Z 204.872,A -85,B 0,C 180,E1 -5912.541,E2 -5912.541} C_VEL
LIN {X 0,Y 502.966,Z 214.362,A -85,B 0,C 180,E1 -5915.682,E2 -5915.682} C_VEL
LIN {X 0,Y 502.851,Z 223.181,A -85,B 0,C 180,E1 -5918.692,E2 -5918.692} C_VEL
LIN {X 0,Y 502.796,Z 230.561,A -85,B 0,C 180,E1 -5921.247,E2 -5921.247} C_VEL
LIN {X 0,Y 502.678,Z 240.078,A -85,B 0,C 180,E1 -5924.595,E2 -5924.595} C_VEL
LIN {X 0,Y 502.665,Z 243.502,A -85,B 0,C 180,E1 -5925.811,E2 -5925.811} C_VEL
LIN {X 0,Y 504.71,Z 254.662,A -85,B 0,C 180,E1 -5926.153,E2 -5926.153} C_VEL
LIN {X 0,Y 504.408,Z 268.306,A -85,B 0,C 180,E1 -5926.658,E2 -5926.658} C_VEL
LIN {X 0,Y 504.091,Z 281.166,A -85,B 0,C 180,E1 -5927.321,E2 -5927.321} C_VEL
LIN {X 0,Y 503.821,Z 293.047,A -85,B 0,C 180,E1 -5928.126,E2 -5928.126} C_VEL
LIN {X 0,Y 503.415,Z 303.729,A -85,B 0,C 180,E1 -5929.035,E2 -5929.035} C_VEL
LIN {X 0,Y 503.066,Z 314.147,A -85,B 0,C 180,E1 -5930.146,E2 -5930.146} C_VEL
LIN {X 0,Y 502.846,Z 321.85,A -85,B 0,C 180,E1 -5931.156,E2 -5931.156} C_VEL
LIN {X 0,Y 502.575,Z 329.378,A -85,B 0,C 180,E1 -5932.366,E2 -5932.366} C_VEL
LIN {X 0,Y 502.445,Z 335.392,A -85,B 0,C 180,E1 -5933.575,E2 -5933.575} C_VEL
LIN {X 0,Y 502.211,Z 340.152,A -85,B 0,C 180,E1 -5934.781,E2 -5934.781} C_VEL
LIN {X 0,Y 502.245,Z 343.777,A -85,B 0,C 180,E1 -5935.988,E2 -5935.988} C_VEL
LIN {X 0,Y 502.247,Z 345.635,A -85,B 0,C 180,E1 -5936.791,E2 -5936.791} C_VEL
LIN {X 0,Y 502.13,Z 347.073,A -85,B 0,C 180,E1 -5937.594,E2 -5937.594} C_VEL
LIN {X 0,Y 502.005,Z 348.675,A -85,B 0,C 180,E1 -5939.198,E2 -5939.198} C_VEL
LIN {X 0,Y 501.999,Z 348.9,A -85,B 0,C 180,E1 -5940,E2 -5940} C_VEL
LIN {X 0,Y 502.003,Z 348.7,A -85,B 0,C 180,E1 -5940.802,E2 -5940.802} C_VEL
LIN {X 0,Y 502.13,Z 347.102,A -85,B 0,C 180,E1 -5942.407,E2 -5942.407} C_VEL
LIN {X 0,Y 502.23,Z 345.702,A -85,B 0,C 180,E1 -5943.209,E2 -5943.209} C_VEL
LIN {X 0,Y 502.235,Z 342.789,A -85,B 0,C 180,E1 -5944.414,E2 -5944.414} C_VEL
LIN {X 0,Y 502.297,Z 338.834,A -85,B 0,C 180,E1 -5945.621,E2 -5945.621} C_VEL
LIN {X 0,Y 502.451,Z 333.188,A -85,B 0,C 180,E1 -5946.94,E2 -5946.94} C_VEL
LIN {X 0,Y 502.646,Z 326.083,A -85,B 0,C 180,E1 -5948.24,E2 -5948.24} C_VEL
LIN {X 0,Y 502.902,Z 317.786,A -85,B 0,C 180,E1 -5949.451,E2 -5949.451} C_VEL
LIN {X 0,Y 503.151,Z 309.253,A -85,B 0,C 180,E1 -5950.462,E2 -5950.462} C_VEL
LIN {X 0,Y 503.537,Z 298.808,A -85,B 0,C 180,E1 -5951.472,E2 -5951.472} C_VEL
LIN {X 0,Y 503.835,Z 288.02,A -85,B 0,C 180,E1 -5952.311,E2 -5952.311} C_VEL
LIN {X 0,Y 504.203,Z 275.137,A -85,B 0,C 180,E1 -5953.092,E2 -5953.092} C_VEL
LIN {X 0,Y 504.545,Z 262.893,A -85,B 0,C 180,E1 -5953.646,E2 -5953.646} C_VEL
LIN {X 0,Y 504.528,Z 253.199,A -85,B 0,C 180,E1 -5953.981,E2 -5953.981} C_VEL
LIN {X 0,Y 502.495,Z 242.457,A -85,B 0,C 180,E1 -5954.323,E2 -5954.323} C_VEL
LIN {X 0,Y 502.667,Z 233.604,A -85,B 0,C 180,E1 -5957.494,E2 -5957.494} C_VEL
LIN {X 0,Y 502.737,Z 225.242,A -85,B 0,C 180,E1 -5960.506,E2 -5960.506} C_VEL
LIN {X 0,Y 502.846,Z 216.999,A -85,B 0,C 180,E1 -5963.474,E2 -5963.474} C_VEL
LIN {X 0,Y 502.947,Z 209.695,A -85,B 0,C 180,E1 -5966.115,E2 -5966.115} C_VEL
LIN {X 0,Y 503.116,Z 202.16,A -85,B 0,C 180,E1 -5968.812,E2 -5968.812} C_VEL
LIN {X 0,Y 503.236,Z 194.466,A -85,B 0,C 180,E1 -5971.58,E2 -5971.58} C_VEL
LIN {X 0,Y 503.328,Z 185.105,A -85,B 0,C 180,E1 -5974.924,E2 -5974.924} C_VEL
LIN {X 0,Y 502.815,Z 180.856,A -85,B 0,C 180,E1 -5976.506,E2 -5976.506} C_VEL
LIN {X 0,Y 502.793,Z 180.857,A -85,B 0,C 180,E1 -5979.754,E2 -5979.754} C_VEL
LIN {X 0,Y 502.809,Z 180.853,A -85,B 0,C 180,E1 -5982.199,E2 -5982.199} C_VEL
LIN {X 0,Y 502.791,Z 180.854,A -85,B 0,C 180,E1 -5985.47,E2 -5985.47} C_VEL
LIN {X 0,Y 502.825,Z 180.853,A -85,B 0,C 180,E1 -5988.934,E2 -5988.934} C_VEL
LIN {X 0,Y 502.792,Z 180.854,A -85,B 0,C 180,E1 -5989.965,E2 -5989.965} C_VEL
LIN {X 0,Y 502.147,Z 180.939,A -85,B 0,C 180,E1 -5990.633,E2 -5990.633} C_VEL
LIN {X 0,Y 499.282,Z 181.294,A -85,B 0,C 180,E1 -5991.718,E2 -5991.718} C_VEL
LIN {X 0,Y 496.84,Z 181.6,A -85,B 0,C 180,E1 -5992.591,E2 -5992.591} C_VEL
LIN {X 0,Y 495.784,Z 181.729,A -85,B 0,C 180,E1 -5993.266,E2 -5993.266} C_VEL
LIN {X 0,Y 495.695,Z 181.741,A -85,B 0,C 180,E1 -5993.495,E2 -5993.495} C_VEL
LIN {X 0,Y 495.755,Z 181.731,A -85,B 0,C 180,E1 -5996.434,E2 -5996.434} C_VEL
LIN {X 0,Y 495.725,Z 181.736,A -85,B 0,C 180,E1 -5999.31,E2 -5999.31} C_VEL
LIN {X 0,Y 495.534,Z 182,A -85,B 0,C 180,E1 -6001.562,E2 -6001.562} C_VEL
LIN {X 0,Y 495.518,Z 184.963,A -85,B 0,C 180,E1 -6003.916,E2 -6003.916} C_VEL
LIN {X 0,Y 495.434,Z 188.351,A -85,B 0,C 180,E1 -6006.596,E2 -6006.596} C_VEL
LIN {X 0,Y 495.371,Z 191.942,A -85,B 0,C 180,E1 -6009.451,E2 -6009.451} C_VEL
LIN {X 0,Y 495.293,Z 196.048,A -85,B 0,C 180,E1 -6012.663,E2 -6012.663} C_VEL
LIN {X 0,Y 495.314,Z 199.409,A -85,B 0,C 180,E1 -6015.202,E2 -6015.202} C_VEL
LIN {X 0,Y 495.303,Z 204.12,A -85,B 0,C 180,E1 -6018.541,E2 -6018.541} C_VEL
LIN {X 0,Y 495.281,Z 208.289,A -85,B 0,C 180,E1 -6021.199,E2 -6021.199} C_VEL
LIN {X 0,Y 496.889,Z 216.024,A -85,B 0,C 180,E1 -6021.51,E2 -6021.51} C_VEL
LIN {X 0,Y 496.819,Z 224.608,A -85,B 0,C 180,E1 -6021.937,E2 -6021.937} C_VEL
LIN {X 0,Y 496.682,Z 233.044,A -85,B 0,C 180,E1 -6022.528,E2 -6022.528} C_VEL
LIN {X 0,Y 496.485,Z 240.258,A -85,B 0,C 180,E1 -6023.19,E2 -6023.19} C_VEL
LIN {X 0,Y 496.335,Z 247.715,A -85,B 0,C 180,E1 -6024.107,E2 -6024.107} C_VEL
LIN {X 0,Y 496.043,Z 253.792,A -85,B 0,C 180,E1 -6025.122,E2 -6025.122} C_VEL
LIN {X 0,Y 495.952,Z 257.432,A -85,B 0,C 180,E1 -6025.936,E2 -6025.936} C_VEL
LIN {X 0,Y 495.741,Z 261.348,A -85,B 0,C 180,E1 -6027.155,E2 -6027.155} C_VEL
LIN {X 0,Y 495.611,Z 263.707,A -85,B 0,C 180,E1 -6028.374,E2 -6028.374} C_VEL
LIN {X 0,Y 495.544,Z 264.541,A -85,B 0,C 180,E1 -6029.186,E2 -6029.186} C_VEL
LIN {X 0,Y 495.519,Z 264.832,A -85,B 0,C 180,E1 -6029.999,E2 -6029.999} C_VEL
LIN {X 0,Y 495.536,Z 264.601,A -85,B 0,C 180,E1 -6030.812,E2 -6030.812} C_VEL
LIN {X 0,Y 495.538,Z 263.841,A -85,B 0,C 180,E1 -6031.624,E2 -6031.624} C_VEL
LIN {X 0,Y 495.613,Z 262.497,A -85,B 0,C 180,E1 -6032.437,E2 -6032.437} C_VEL
LIN {X 0,Y 495.871,Z 259.248,A -85,B 0,C 180,E1 -6033.656,E2 -6033.656} C_VEL
LIN {X 0,Y 495.973,Z 256.147,A -85,B 0,C 180,E1 -6034.469,E2 -6034.469} C_VEL
LIN {X 0,Y 496.253,Z 250.944,A -85,B 0,C 180,E1 -6035.484,E2 -6035.484} C_VEL
LIN {X 0,Y 496.401,Z 245.386,A -85,B 0,C 180,E1 -6036.298,E2 -6036.298} C_VEL
LIN {X 0,Y 496.504,Z 239.151,A -85,B 0,C 180,E1 -6037.011,E2 -6037.011} C_VEL
LIN {X 0,Y 496.712,Z 232.887,A -85,B 0,C 180,E1 -6037.574,E2 -6037.574} C_VEL
LIN {X 0,Y 496.788,Z 224.986,A -85,B 0,C 180,E1 -6038.132,E2 -6038.132} C_VEL
LIN {X 0,Y 496.835,Z 215.791,A -85,B 0,C 180,E1 -6038.592,E2 -6038.592} C_VEL
LIN {X 0,Y 495.239,Z 208.161,A -85,B 0,C 180,E1 -6038.902,E2 -6038.902} C_VEL
LIN {X 0,Y 495.337,Z 203.811,A -85,B 0,C 180,E1 -6041.763,E2 -6041.763} C_VEL
LIN {X 0,Y 495.307,Z 198.935,A -85,B 0,C 180,E1 -6045.232,E2 -6045.232} C_VEL
LIN {X 0,Y 495.323,Z 195.086,A -85,B 0,C 180,E1 -6048.188,E2 -6048.188} C_VEL
LIN {X 0,Y 495.365,Z 191.784,A -85,B 0,C 180,E1 -6050.773,E2 -6050.773} C_VEL
LIN {X 0,Y 495.429,Z 188.515,A -85,B 0,C 180,E1 -6053.402,E2 -6053.402} C_VEL
LIN {X 0,Y 495.511,Z 185.141,A -85,B 0,C 180,E1 -6056.082,E2 -6056.082} C_VEL
LIN {X 0,Y 495.547,Z 181.762,A -85,B 0,C 180,E1 -6058.828,E2 -6058.828} C_VEL
LIN {X 0,Y 495.718,Z 181.734,A -85,B 0,C 180,E1 -6060.688,E2 -6060.688} C_VEL
LIN {X 0,Y 495.756,Z 181.735,A -85,B 0,C 180,E1 -6063.563,E2 -6063.563} C_VEL
LIN {X 0,Y 495.728,Z 181.732,A -85,B 0,C 180,E1 -6066.542,E2 -6066.542} C_VEL
LIN {X 0,Y 495.751,Z 181.732,A -85,B 0,C 180,E1 -6069.637,E2 -6069.637} C_VEL
LIN {X 0,Y 495.734,Z 181.732,A -85,B 0,C 180,E1 -6072.506,E2 -6072.506} C_VEL
LIN {X 0,Y 495.742,Z 181.736,A -85,B 0,C 180,E1 -6075.138,E2 -6075.138} C_VEL
LIN {X 0,Y 495.751,Z 181.73,A -85,B 0,C 180,E1 -6078.218,E2 -6078.218} C_VEL
LIN {X 0,Y 495.744,Z 181.73,A -85,B 0,C 180,E1 -6081.408,E2 -6081.408} C_VEL
LIN {X 0,Y 495.75,Z 181.734,A -85,B 0,C 180,E1 -6084.462,E2 -6084.462} C_VEL
LIN {X 0,Y 495.761,Z 181.726,A -85,B 0,C 180,E1 -6087.405,E2 -6087.405} C_VEL
LIN {X 0,Y 495.773,Z 181.73,A -85,B 0,C 180,E1 -6090.254,E2 -6090.254} C_VEL
LIN {X 0,Y 495.824,Z 181.719,A -85,B 0,C 180,E1 -6093.247,E2 -6093.247} C_VEL
LIN {X 0,Y 495.742,Z 181.729,A -85,B 0,C 180,E1 -6095.724,E2 -6095.724} C_VEL
LIN {X 0,Y 495.734,Z 181.731,A -85,B 0,C 180,E1 -6098.371,E2 -6098.371} C_VEL
LIN {X 0,Y 495.774,Z 181.724,A -85,B 0,C 180,E1 -6100.971,E2 -6100.971} C_VEL
LIN {X 0,Y 495.771,Z 181.731,A -85,B 0,C 180,E1 -6103.53,E2 -6103.53} C_VEL
LIN {X 0,Y 495.783,Z 181.726,A -85,B 0,C 180,E1 -6106.055,E2 -6106.055} C_VEL
LIN {X 0,Y 495.844,Z 181.716,A -85,B 0,C 180,E1 -6108.555,E2 -6108.555} C_VEL
LIN {X 0,Y 495.863,Z 181.716,A -85,B 0,C 180,E1 -6111.852,E2 -6111.852} C_VEL
LIN {X 0,Y 495.879,Z 181.71,A -85,B 0,C 180,E1 -6114.306,E2 -6114.306} C_VEL
LIN {X 0,Y 495.979,Z 181.701,A -85,B 0,C 180,E1 -6117.564,E2 -6117.564} C_VEL
LIN {X 0,Y 495.983,Z 181.695,A -85,B 0,C 180,E1 -6120,E2 -6120} C_VEL
LIN {X 0,Y 495.979,Z 181.702,A -85,B 0,C 180,E1 -6122.436,E2 -6122.436} C_VEL
LIN {X 0,Y 495.874,Z 181.711,A -85,B 0,C 180,E1 -6125.694,E2 -6125.694} C_VEL
LIN {X 0,Y 495.859,Z 181.717,A -85,B 0,C 180,E1 -6128.148,E2 -6128.148} C_VEL
LIN {X 0,Y 495.838,Z 181.718,A -85,B 0,C 180,E1 -6131.446,E2 -6131.446} C_VEL
LIN {X 0,Y 495.776,Z 181.728,A -85,B 0,C 180,E1 -6134.783,E2 -6134.783} C_VEL
LIN {X 0,Y 495.767,Z 181.731,A -85,B 0,C 180,E1 -6138.172,E2 -6138.172} C_VEL
LIN {X 0,Y 495.762,Z 181.728,A -85,B 0,C 180,E1 -6140.757,E2 -6140.757} C_VEL
LIN {X 0,Y 495.726,Z 181.734,A -85,B 0,C 180,E1 -6143.388,E2 -6143.388} C_VEL
LIN {X 0,Y 495.726,Z 181.732,A -85,B 0,C 180,E1 -6146.73,E2 -6146.73} C_VEL
LIN {X 0,Y 495.745,Z 181.736,A -85,B 0,C 180,E1 -6149.748,E2 -6149.748} C_VEL
LIN {X 0,Y 495.756,Z 181.728,A -85,B 0,C 180,E1 -6152.595,E2 -6152.595} C_VEL
LIN {X 0,Y 495.733,Z 181.737,A -85,B 0,C 180,E1 -6155.539,E2 -6155.539} C_VEL
LIN {X 0,Y 495.748,Z 181.734,A -85,B 0,C 180,E1 -6158.768,E2 -6158.768} C_VEL
LIN {X 0,Y 495.736,Z 181.732,A -85,B 0,C 180,E1 -6161.783,E2 -6161.783} C_VEL
LIN {X 0,Y 495.729,Z 181.736,A -85,B 0,C 180,E1 -6165.142,E2 -6165.142} C_VEL
LIN {X 0,Y 495.749,Z 181.726,A -85,B 0,C 180,E1 -6168.22,E2 -6168.22} C_VEL
LIN {X 0,Y 495.744,Z 181.733,A -85,B 0,C 180,E1 -6171.41,E2 -6171.41} C_VEL
LIN {X 0,Y 495.743,Z 181.735,A -85,B 0,C 180,E1 -6174.464,E2 -6174.464} C_VEL
LIN {X 0,Y 495.783,Z 181.779,A -85,B 0,C 180,E1 -6176.635,E2 -6176.635} C_VEL
LIN {X 0,Y 498.625,Z 194.091,A -85,B 0,C 180,E1 -6179.292,E2 -6179.292} C_VEL
LIN {X 0,Y 499.415,Z 199.008,A -85,B 0,C 180,E1 -6180.262,E2 -6180.262} C_VEL
LIN {X 0,Y 498.608,Z 213.875,A -85,B 0,C 180,E1 -6182.9,E2 -6182.9} C_VEL
LIN {X 0,Y 497.717,Z 232.66,A -85,B 0,C 180,E1 -6186.072,E2 -6186.072} C_VEL
LIN {X 0,Y 496.977,Z 252.257,A -85,B 0,C 180,E1 -6189.297,E2 -6189.297} C_VEL
LIN {X 0,Y 496.398,Z 269.213,A -85,B 0,C 180,E1 -6192.066,E2 -6192.066} C_VEL
LIN {X 0,Y 495.889,Z 289.479,A -85,B 0,C 180,E1 -6195.431,E2 -6195.431} C_VEL
LIN {X 0,Y 495.832,Z 291.033,A -85,B 0,C 180,E1 -6195.692,E2 -6195.692} C_VEL
LIN {X 0,Y 497.173,Z 305.858,A -85,B 0,C 180,E1 -6196.044,E2 -6196.044} C_VEL
LIN {X 0,Y 497.019,Z 318.312,A -85,B 0,C 180,E1 -6196.457,E2 -6196.457} C_VEL
LIN {X 0,Y 496.715,Z 330.476,A -85,B 0,C 180,E1 -6197.021,E2 -6197.021} C_VEL
LIN {X 0,Y 496.384,Z 342.283,A -85,B 0,C 180,E1 -6197.74,E2 -6197.74} C_VEL
LIN {X 0,Y 496.06,Z 354.039,A -85,B 0,C 180,E1 -6198.664,E2 -6198.664} C_VEL
LIN {X 0,Y 495.794,Z 363.515,A -85,B 0,C 180,E1 -6199.589,E2 -6199.589} C_VEL
LIN {X 0,Y 495.561,Z 372.157,A -85,B 0,C 180,E1 -6200.615,E2 -6200.615} C_VEL
LIN {X 0,Y 495.366,Z 380.546,A -85,B 0,C 180,E1 -6201.845,E2 -6201.845} C_VEL
LIN {X 0,Y 495.233,Z 387.468,A -85,B 0,C 180,E1 -6203.114,E2 -6203.114} C_VEL
LIN {X 0,Y 495.193,Z 392.599,A -85,B 0,C 180,E1 -6204.3,E2 -6204.3} C_VEL
LIN {X 0,Y 495.187,Z 396.723,A -85,B 0,C 180,E1 -6205.524,E2 -6205.524} C_VEL
LIN {X 0,Y 495.159,Z 399.76,A -85,B 0,C 180,E1 -6206.746,E2 -6206.746} C_VEL
LIN {X 0,Y 495.143,Z 401.206,A -85,B 0,C 180,E1 -6207.561,E2 -6207.561} C_VEL
LIN {X 0,Y 495.09,Z 402.228,A -85,B 0,C 180,E1 -6208.374,E2 -6208.374} C_VEL
LIN {X 0,Y 495.106,Z 402.841,A -85,B 0,C 180,E1 -6209.188,E2 -6209.188} C_VEL
LIN {X 0,Y 495.125,Z 403.049,A -85,B 0,C 180,E1 -6210.001,E2 -6210.001} C_VEL
LIN {X 0,Y 495.108,Z 402.795,A -85,B 0,C 180,E1 -6210.814,E2 -6210.814} C_VEL
LIN {X 0,Y 495.143,Z 401.111,A -85,B 0,C 180,E1 -6212.442,E2 -6212.442} C_VEL
LIN {X 0,Y 495.189,Z 399.611,A -85,B 0,C 180,E1 -6213.255,E2 -6213.255} C_VEL
LIN {X 0,Y 495.202,Z 396.523,A -85,B 0,C 180,E1 -6214.478,E2 -6214.478} C_VEL
LIN {X 0,Y 495.216,Z 392.324,A -85,B 0,C 180,E1 -6215.702,E2 -6215.702} C_VEL
LIN {X 0,Y 495.266,Z 385.952,A -85,B 0,C 180,E1 -6217.113,E2 -6217.113} C_VEL
LIN {X 0,Y 495.425,Z 378.785,A -85,B 0,C 180,E1 -6218.362,E2 -6218.362} C_VEL
LIN {X 0,Y 495.584,Z 369.936,A -85,B 0,C 180,E1 -6219.593,E2 -6219.593} C_VEL
LIN {X 0,Y 495.87,Z 359.833,A -85,B 0,C 180,E1 -6220.722,E2 -6220.722} C_VEL
LIN {X 0,Y 496.177,Z 348.522,A -85,B 0,C 180,E1 -6221.726,E2 -6221.726} C_VEL
LIN {X 0,Y 496.441,Z 338.445,A -85,B 0,C 180,E1 -6222.448,E2 -6222.448} C_VEL
LIN {X 0,Y 496.78,Z 326.354,A -85,B 0,C 180,E1 -6223.135,E2 -6223.135} C_VEL
LIN {X 0,Y 497.04,Z 313.544,A -85,B 0,C 180,E1 -6223.675,E2 -6223.675} C_VEL
LIN {X 0,Y 497.02,Z 304.96,A -85,B 0,C 180,E1 -6223.949,E2 -6223.949} C_VEL
LIN {X 0,Y 495.836,Z 291.032,A -85,B 0,C 180,E1 -6224.31,E2 -6224.31} C_VEL
LIN {X 0,Y 496.342,Z 271.762,A -85,B 0,C 180,E1 -6227.512,E2 -6227.512} C_VEL
LIN {X 0,Y 497.131,Z 248.901,A -85,B 0,C 180,E1 -6231.256,E2 -6231.256} C_VEL
LIN {X 0,Y 497.787,Z 231.198,A -85,B 0,C 180,E1 -6234.17,E2 -6234.17} C_VEL
LIN {X 0,Y 498.658,Z 212.192,A -85,B 0,C 180,E1 -6237.388,E2 -6237.388} C_VEL
LIN {X 0,Y 499.425,Z 198.93,A -85,B 0,C 180,E1 -6239.739,E2 -6239.739} C_VEL
LIN {X 0,Y 498.008,Z 191.432,A -85,B 0,C 180,E1 -6241.259,E2 -6241.259} C_VEL
LIN {X 0,Y 495.736,Z 181.741,A -85,B 0,C 180,E1 -6243.416,E2 -6243.416} C_VEL
LIN {X 0,Y 495.715,Z 181.739,A -85,B 0,C 180,E1 -6246.087,E2 -6246.087} C_VEL
LIN {X 0,Y 495.763,Z 181.733,A -85,B 0,C 180,E1 -6248.768,E2 -6248.768} C_VEL
LIN {X 0,Y 495.761,Z 181.732,A -85,B 0,C 180,E1 -6251.782,E2 -6251.782} C_VEL
LIN {X 0,Y 495.742,Z 181.734,A -85,B 0,C 180,E1 -6255.141,E2 -6255.141} C_VEL
LIN {X 0,Y 495.761,Z 181.731,A -85,B 0,C 180,E1 -6258.219,E2 -6258.219} C_VEL
LIN {X 0,Y 495.75,Z 181.735,A -85,B 0,C 180,E1 -6261.408,E2 -6261.408} C_VEL
LIN {X 0,Y 495.736,Z 181.74,A -85,B 0,C 180,E1 -6264.915,E2 -6264.915} C_VEL
LIN {X 0,Y 496.141,Z 185.084,A -85,B 0,C 180,E1 -6265.977,E2 -6265.977} C_VEL
LIN {X 0,Y 496.053,Z 194.6,A -85,B 0,C 180,E1 -6268.86,E2 -6268.86} C_VEL
LIN {X 0,Y 496,Z 204.886,A -85,B 0,C 180,E1 -6272.122,E2 -6272.122} C_VEL
LIN {X 0,Y 495.931,Z 212.968,A -85,B 0,C 180,E1 -6274.84,E2 -6274.84} C_VEL
LIN {X 0,Y 495.871,Z 220.89,A -85,B 0,C 180,E1 -6277.501,E2 -6277.501} C_VEL
LIN {X 0,Y 495.814,Z 229.657,A -85,B 0,C 180,E1 -6280.543,E2 -6280.543} C_VEL
LIN {X 0,Y 495.678,Z 238.128,A -85,B 0,C 180,E1 -6283.527,E2 -6283.527} C_VEL
LIN {X 0,Y 495.651,Z 244.039,A -85,B 0,C 180,E1 -6285.606,E2 -6285.606} C_VEL
LIN {X 0,Y 497.836,Z 255.008,A -85,B 0,C 180,E1 -6285.958,E2 -6285.958} C_VEL
LIN {X 0,Y 497.524,Z 268.581,A -85,B 0,C 180,E1 -6286.47,E2 -6286.47} C_VEL
LIN {X 0,Y 497.175,Z 280.488,A -85,B 0,C 180,E1 -6287.083,E2 -6287.083} C_VEL
LIN {X 0,Y 496.916,Z 291.971,A -85,B 0,C 180,E1 -6287.855,E2 -6287.855} C_VEL
LIN {X 0,Y 496.497,Z 302.954,A -85,B 0,C 180,E1 -6288.777,E2 -6288.777} C_VEL
LIN {X 0,Y 496.141,Z 312.736,A -85,B 0,C 180,E1 -6289.801,E2 -6289.801} C_VEL
LIN {X 0,Y 495.834,Z 322.176,A -85,B 0,C 180,E1 -6291.03,E2 -6291.03} C_VEL
LIN {X 0,Y 495.53,Z 329.725,A -85,B 0,C 180,E1 -6292.257,E2 -6292.257} C_VEL
LIN {X 0,Y 495.374,Z 335.754,A -85,B 0,C 180,E1 -6293.483,E2 -6293.483} C_VEL
LIN {X 0,Y 495.15,Z 340.525,A -85,B 0,C 180,E1 -6294.706,E2 -6294.706} C_VEL
LIN {X 0,Y 495.184,Z 344.158,A -85,B 0,C 180,E1 -6295.931,E2 -6295.931} C_VEL
LIN {X 0,Y 495.161,Z 346.022,A -85,B 0,C 180,E1 -6296.745,E2 -6296.745} C_VEL
LIN {X 0,Y 495.068,Z 347.461,A -85,B 0,C 180,E1 -6297.559,E2 -6297.559} C_VEL
LIN {X 0,Y 494.924,Z 349.064,A -85,B 0,C 180,E1 -6299.186,E2 -6299.186} C_VEL
LIN {X 0,Y 494.916,Z 349.286,A -85,B 0,C 180,E1 -6300,E2 -6300} C_VEL
LIN {X 0,Y 494.922,Z 349.082,A -85,B 0,C 180,E1 -6300.814,E2 -6300.814} C_VEL
LIN {X 0,Y 495.067,Z 347.469,A -85,B 0,C 180,E1 -6302.441,E2 -6302.441} C_VEL
LIN {X 0,Y 495.146,Z 346.065,A -85,B 0,C 180,E1 -6303.255,E2 -6303.255} C_VEL
LIN {X 0,Y 495.165,Z 343.136,A -85,B 0,C 180,E1 -6304.477,E2 -6304.477} C_VEL
LIN {X 0,Y 495.248,Z 339.164,A -85,B 0,C 180,E1 -6305.701,E2 -6305.701} C_VEL
LIN {X 0,Y 495.411,Z 333.14,A -85,B 0,C 180,E1 -6307.11,E2 -6307.11} C_VEL
LIN {X 0,Y 495.63,Z 326.36,A -85,B 0,C 180,E1 -6308.357,E2 -6308.357} C_VEL
LIN {X 0,Y 495.895,Z 318.027,A -85,B 0,C 180,E1 -6309.586,E2 -6309.586} C_VEL
LIN {X 0,Y 496.165,Z 309.468,A -85,B 0,C 180,E1 -6310.611,E2 -6310.611} C_VEL
LIN {X 0,Y 496.591,Z 298.997,A -85,B 0,C 180,E1 -6311.635,E2 -6311.635} C_VEL
LIN {X 0,Y 496.893,Z 288.779,A -85,B 0,C 180,E1 -6312.443,E2 -6312.443} C_VEL
LIN {X 0,Y 497.254,Z 277.107,A -85,B 0,C 180,E1 -6313.174,E2 -6313.174} C_VEL
LIN {X 0,Y 497.631,Z 264.27,A -85,B 0,C 180,E1 -6313.788,E2 -6313.788} C_VEL
LIN {X 0,Y 497.616,Z 254.087,A -85,B 0,C 180,E1 -6314.153,E2 -6314.153} C_VEL
LIN {X 0,Y 495.477,Z 242.804,A -85,B 0,C 180,E1 -6314.504,E2 -6314.504} C_VEL
LIN {X 0,Y 495.591,Z 234.98,A -85,B 0,C 180,E1 -6317.326,E2 -6317.326} C_VEL
LIN {X 0,Y 495.724,Z 226.825,A -85,B 0,C 180,E1 -6320.272,E2 -6320.272} C_VEL
LIN {X 0,Y 495.806,Z 218.249,A -85,B 0,C 180,E1 -6323.384,E2 -6323.384} C_VEL
LIN {X 0,Y 495.931,Z 210.852,A -85,B 0,C 180,E1 -6326.06,E2 -6326.06} C_VEL
LIN {X 0,Y 496.098,Z 203.299,A -85,B 0,C 180,E1 -6328.794,E2 -6328.794} C_VEL
LIN {X 0,Y 496.217,Z 195.537,A -85,B 0,C 180,E1 -6331.604,E2 -6331.604} C_VEL
LIN {X 0,Y 496.307,Z 186.679,A -85,B 0,C 180,E1 -6334.782,E2 -6334.782} C_VEL
LIN {X 0,Y 495.791,Z 181.73,A -85,B 0,C 180,E1 -6336.602,E2 -6336.602} C_VEL
LIN {X 0,Y 495.761,Z 181.734,A -85,B 0,C 180,E1 -6339.638,E2 -6339.638} C_VEL
LIN {X 0,Y 495.739,Z 181.736,A -85,B 0,C 180,E1 -6342.506,E2 -6342.506} C_VEL
LIN {X 0,Y 495.743,Z 181.73,A -85,B 0,C 180,E1 -6345.141,E2 -6345.141} C_VEL
LIN {X 0,Y 495.761,Z 181.73,A -85,B 0,C 180,E1 -6348.219,E2 -6348.219} C_VEL
LIN {X 0,Y 495.75,Z 181.733,A -85,B 0,C 180,E1 -6351.234,E2 -6351.234} C_VEL
LIN {X 0,Y 495.695,Z 181.741,A -85,B 0,C 180,E1 -6353.495,E2 -6353.495} C_VEL
LIN {X 0,Y 495.035,Z 181.826,A -85,B 0,C 180,E1 -6354.173,E2 -6354.173} C_VEL
LIN {X 0,Y 492.235,Z 182.177,A -85,B 0,C 180,E1 -6355.276,E2 -6355.276} C_VEL
LIN {X 0,Y 489.857,Z 182.472,A -85,B 0,C 180,E1 -6356.165,E2 -6356.165} C_VEL
LIN {X 0,Y 488.817,Z 182.598,A -85,B 0,C 180,E1 -6356.851,E2 -6356.851} C_VEL
LIN {X 0,Y 488.721,Z 182.608,A -85,B 0,C 180,E1 -6357.083,E2 -6357.083} C_VEL
LIN {X 0,Y 488.668,Z 182.615,A -85,B 0,C 180,E1 -6359.776,E2 -6359.776} C_VEL
LIN {X 0,Y 488.504,Z 182.639,A -85,B 0,C 180,E1 -6361.354,E2 -6361.354} C_VEL
LIN {X 0,Y 488.446,Z 186.452,A -85,B 0,C 180,E1 -6364.426,E2 -6364.426} C_VEL
LIN {X 0,Y 488.367,Z 189.85,A -85,B 0,C 180,E1 -6367.135,E2 -6367.135} C_VEL
LIN {X 0,Y 488.304,Z 193.178,A -85,B 0,C 180,E1 -6369.791,E2 -6369.791} C_VEL
LIN {X 0,Y 488.246,Z 196.519,A -85,B 0,C 180,E1 -6372.404,E2 -6372.404} C_VEL
LIN {X 0,Y 488.247,Z 199.921,A -85,B 0,C 180,E1 -6374.982,E2 -6374.982} C_VEL
LIN {X 0,Y 488.274,Z 204.697,A -85,B 0,C 180,E1 -6378.374,E2 -6378.374} C_VEL
LIN {X 0,Y 488.204,Z 208.741,A -85,B 0,C 180,E1 -6381.018,E2 -6381.018} C_VEL
LIN {X 0,Y 489.941,Z 217.782,A -85,B 0,C 180,E1 -6381.388,E2 -6381.388} C_VEL
LIN {X 0,Y 489.853,Z 227.127,A -85,B 0,C 180,E1 -6381.892,E2 -6381.892} C_VEL
LIN {X 0,Y 489.732,Z 235.206,A -85,B 0,C 180,E1 -6382.49,E2 -6382.49} C_VEL
LIN {X 0,Y 489.505,Z 242.488,A -85,B 0,C 180,E1 -6383.196,E2 -6383.196} C_VEL
LIN {X 0,Y 489.378,Z 248.873,A -85,B 0,C 180,E1 -6384.023,E2 -6384.023} C_VEL
LIN {X 0,Y 489.16,Z 253.844,A -85,B 0,C 180,E1 -6384.847,E2 -6384.847} C_VEL
LIN {X 0,Y 488.973,Z 258.493,A -85,B 0,C 180,E1 -6385.878,E2 -6385.878} C_VEL
LIN {X 0,Y 488.739,Z 262.367,A -85,B 0,C 180,E1 -6387.114,E2 -6387.114} C_VEL
LIN {X 0,Y 488.599,Z 264.697,A -85,B 0,C 180,E1 -6388.35,E2 -6388.35} C_VEL
LIN {X 0,Y 488.527,Z 265.519,A -85,B 0,C 180,E1 -6389.175,E2 -6389.175} C_VEL
LIN {X 0,Y 488.5,Z 265.805,A -85,B 0,C 180,E1 -6389.999,E2 -6389.999} C_VEL
LIN {X 0,Y 488.519,Z 265.577,A -85,B 0,C 180,E1 -6390.823,E2 -6390.823} C_VEL
LIN {X 0,Y 488.534,Z 264.824,A -85,B 0,C 180,E1 -6391.648,E2 -6391.648} C_VEL
LIN {X 0,Y 488.601,Z 263.499,A -85,B 0,C 180,E1 -6392.472,E2 -6392.472} C_VEL
LIN {X 0,Y 488.889,Z 260.284,A -85,B 0,C 180,E1 -6393.708,E2 -6393.708} C_VEL
LIN {X 0,Y 488.986,Z 257.22,A -85,B 0,C 180,E1 -6394.533,E2 -6394.533} C_VEL
LIN {X 0,Y 489.279,Z 252.064,A -85,B 0,C 180,E1 -6395.563,E2 -6395.563} C_VEL
LIN {X 0,Y 489.448,Z 246.574,A -85,B 0,C 180,E1 -6396.388,E2 -6396.388} C_VEL
LIN {X 0,Y 489.567,Z 240.395,A -85,B 0,C 180,E1 -6397.111,E2 -6397.111} C_VEL
LIN {X 0,Y 489.754,Z 234.21,A -85,B 0,C 180,E1 -6397.683,E2 -6397.683} C_VEL
LIN {X 0,Y 489.875,Z 226.433,A -85,B 0,C 180,E1 -6398.247,E2 -6398.247} C_VEL
LIN {X 0,Y 489.982,Z 217.506,A -85,B 0,C 180,E1 -6398.713,E2 -6398.713} C_VEL
LIN {X 0,Y 488.198,Z 208.726,A -85,B 0,C 180,E1 -6399.084,E2 -6399.084} C_VEL
LIN {X 0,Y 488.289,Z 204.532,A -85,B 0,C 180,E1 -6401.837,E2 -6401.837} C_VEL
LIN {X 0,Y 488.268,Z 199.602,A -85,B 0,C 180,E1 -6405.338,E2 -6405.338} C_VEL
LIN {X 0,Y 488.273,Z 195.55,A -85,B 0,C 180,E1 -6408.46,E2 -6408.46} C_VEL
LIN {X 0,Y 488.302,Z 192.197,A -85,B 0,C 180,E1 -6411.088,E2 -6411.088} C_VEL
LIN {X 0,Y 488.382,Z 188.875,A -85,B 0,C 180,E1 -6413.76,E2 -6413.76} C_VEL
LIN {X 0,Y 488.495,Z 184.946,A -85,B 0,C 180,E1 -6416.874,E2 -6416.874} C_VEL
LIN {X 0,Y 488.51,Z 182.695,A -85,B 0,C 180,E1 -6418.647,E2 -6418.647} C_VEL
LIN {X 0,Y 488.673,Z 182.614,A -85,B 0,C 180,E1 -6421.18,E2 -6421.18} C_VEL
LIN {X 0,Y 488.729,Z 182.606,A -85,B 0,C 180,E1 -6424.111,E2 -6424.111} C_VEL
LIN {X 0,Y 488.677,Z 182.615,A -85,B 0,C 180,E1 -6427.157,E2 -6427.157} C_VEL
LIN {X 0,Y 488.712,Z 182.606,A -85,B 0,C 180,E1 -6430.343,E2 -6430.343} C_VEL
LIN {X 0,Y 488.709,Z 182.61,A -85,B 0,C 180,E1 -6432.826,E2 -6432.826} C_VEL
LIN {X 0,Y 488.693,Z 182.607,A -85,B 0,C 180,E1 -6435.975,E2 -6435.975} C_VEL
LIN {X 0,Y 488.702,Z 182.611,A -85,B 0,C 180,E1 -6438.584,E2 -6438.584} C_VEL
LIN {X 0,Y 488.697,Z 182.612,A -85,B 0,C 180,E1 -6440.946,E2 -6440.946} C_VEL
LIN {X 0,Y 488.678,Z 182.609,A -85,B 0,C 180,E1 -6443.868,E2 -6443.868} C_VEL
LIN {X 0,Y 488.731,Z 182.605,A -85,B 0,C 180,E1 -6446.876,E2 -6446.876} C_VEL
LIN {X 0,Y 488.725,Z 182.604,A -85,B 0,C 180,E1 -6449.781,E2 -6449.781} C_VEL
LIN {X 0,Y 488.789,Z 182.596,A -85,B 0,C 180,E1 -6453.054,E2 -6453.054} C_VEL
LIN {X 0,Y 488.684,Z 182.614,A -85,B 0,C 180,E1 -6456.254,E2 -6456.254} C_VEL
LIN {X 0,Y 488.735,Z 182.601,A -85,B 0,C 180,E1 -6459.175,E2 -6459.175} C_VEL
LIN {X 0,Y 488.748,Z 182.605,A -85,B 0,C 180,E1 -6461.627,E2 -6461.627} C_VEL
LIN {X 0,Y 488.751,Z 182.597,A -85,B 0,C 180,E1 -6464.999,E2 -6464.999} C_VEL
LIN {X 0,Y 488.797,Z 182.594,A -85,B 0,C 180,E1 -6468.387,E2 -6468.387} C_VEL
LIN {X 0,Y 488.808,Z 182.596,A -85,B 0,C 180,E1 -6471.733,E2 -6471.733} C_VEL
LIN {X 0,Y 488.837,Z 182.587,A -85,B 0,C 180,E1 -6474.224,E2 -6474.224} C_VEL
LIN {X 0,Y 488.947,Z 182.578,A -85,B 0,C 180,E1 -6477.529,E2 -6477.529} C_VEL
LIN {X 0,Y 488.943,Z 182.578,A -85,B 0,C 180,E1 -6480.824,E2 -6480.824} C_VEL
LIN {X 0,Y 488.946,Z 182.579,A -85,B 0,C 180,E1 -6482.471,E2 -6482.471} C_VEL
LIN {X 0,Y 488.833,Z 182.589,A -85,B 0,C 180,E1 -6485.776,E2 -6485.776} C_VEL
LIN {X 0,Y 488.803,Z 182.597,A -85,B 0,C 180,E1 -6488.267,E2 -6488.267} C_VEL
LIN {X 0,Y 488.792,Z 182.596,A -85,B 0,C 180,E1 -6491.613,E2 -6491.613} C_VEL
LIN {X 0,Y 488.749,Z 182.602,A -85,B 0,C 180,E1 -6495.001,E2 -6495.001} C_VEL
LIN {X 0,Y 488.733,Z 182.607,A -85,B 0,C 180,E1 -6498.443,E2 -6498.443} C_VEL
LIN {X 0,Y 488.694,Z 182.608,A -85,B 0,C 180,E1 -6501.071,E2 -6501.071} C_VEL
LIN {X 0,Y 488.657,Z 182.619,A -85,B 0,C 180,E1 -6503.747,E2 -6503.747} C_VEL
LIN {X 0,Y 488.684,Z 182.61,A -85,B 0,C 180,E1 -6506.922,E2 -6506.922} C_VEL
LIN {X 0,Y 488.706,Z 182.608,A -85,B 0,C 180,E1 -6510.221,E2 -6510.221} C_VEL
LIN {X 0,Y 488.72,Z 182.61,A -85,B 0,C 180,E1 -6513.484,E2 -6513.484} C_VEL
LIN {X 0,Y 488.663,Z 182.612,A -85,B 0,C 180,E1 -6516.354,E2 -6516.354} C_VEL
LIN {X 0,Y 488.684,Z 182.613,A -85,B 0,C 180,E1 -6519.256,E2 -6519.256} C_VEL
LIN {X 0,Y 488.68,Z 182.613,A -85,B 0,C 180,E1 -6522.527,E2 -6522.527} C_VEL
LIN {X 0,Y 488.693,Z 182.612,A -85,B 0,C 180,E1 -6525.198,E2 -6525.198} C_VEL
LIN {X 0,Y 488.7,Z 182.606,A -85,B 0,C 180,E1 -6528.401,E2 -6528.401} C_VEL
LIN {X 0,Y 488.698,Z 182.609,A -85,B 0,C 180,E1 -6530.949,E2 -6530.949} C_VEL
LIN {X 0,Y 488.672,Z 182.613,A -85,B 0,C 180,E1 -6533.869,E2 -6533.869} C_VEL
LIN {X 0,Y 488.738,Z 182.67,A -85,B 0,C 180,E1 -6536.282,E2 -6536.282} C_VEL
LIN {X 0,Y 491.814,Z 195.981,A -85,B 0,C 180,E1 -6539.213,E2 -6539.213} C_VEL
LIN {X 0,Y 492.569,Z 200.074,A -85,B 0,C 180,E1 -6540.042,E2 -6540.042} C_VEL
LIN {X 0,Y 491.984,Z 210.12,A -85,B 0,C 180,E1 -6541.876,E2 -6541.876} C_VEL
LIN {X 0,Y 491.069,Z 226.896,A -85,B 0,C 180,E1 -6544.802,E2 -6544.802} C_VEL
LIN {X 0,Y 490.318,Z 243.902,A -85,B 0,C 180,E1 -6547.678,E2 -6547.678} C_VEL
LIN {X 0,Y 489.632,Z 263.305,A -85,B 0,C 180,E1 -6550.917,E2 -6550.917} C_VEL
LIN {X 0,Y 488.949,Z 282.498,A -85,B 0,C 180,E1 -6554.152,E2 -6554.152} C_VEL
LIN {X 0,Y 488.785,Z 290.232,A -85,B 0,C 180,E1 -6555.481,E2 -6555.481} C_VEL
LIN {X 0,Y 490.144,Z 305.37,A -85,B 0,C 180,E1 -6555.84,E2 -6555.84} C_VEL
LIN {X 0,Y 490.107,Z 317.794,A -85,B 0,C 180,E1 -6556.262,E2 -6556.262} C_VEL
LIN {X 0,Y 489.736,Z 329.975,A -85,B 0,C 180,E1 -6556.833,E2 -6556.833} C_VEL
LIN {X 0,Y 489.431,Z 341.807,A -85,B 0,C 180,E1 -6557.563,E2 -6557.563} C_VEL
LIN {X 0,Y 489.04,Z 353.571,A -85,B 0,C 180,E1 -6558.499,E2 -6558.499} C_VEL
LIN {X 0,Y 488.763,Z 363.068,A -85,B 0,C 180,E1 -6559.437,E2 -6559.437} C_VEL
LIN {X 0,Y 488.507,Z 371.728,A -85,B 0,C 180,E1 -6560.478,E2 -6560.478} C_VEL
LIN {X 0,Y 488.311,Z 380.122,A -85,B 0,C 180,E1 -6561.726,E2 -6561.726} C_VEL
LIN {X 0,Y 488.149,Z 386.853,A -85,B 0,C 180,E1 -6562.972,E2 -6562.972} C_VEL
LIN {X 0,Y 488.107,Z 392.203,A -85,B 0,C 180,E1 -6564.217,E2 -6564.217} C_VEL
LIN {X 0,Y 488.083,Z 396.335,A -85,B 0,C 180,E1 -6565.459,E2 -6565.459} C_VEL
LIN {X 0,Y 488.081,Z 399.374,A -85,B 0,C 180,E1 -6566.699,E2 -6566.699} C_VEL
LIN {X 0,Y 488.074,Z 400.829,A -85,B 0,C 180,E1 -6567.525,E2 -6567.525} C_VEL
LIN {X 0,Y 488.011,Z 401.846,A -85,B 0,C 180,E1 -6568.351,E2 -6568.351} C_VEL
LIN {X 0,Y 488.017,Z 402.458,A -85,B 0,C 180,E1 -6569.176,E2 -6569.176} C_VEL
LIN {X 0,Y 488.036,Z 402.665,A -85,B 0,C 180,E1 -6570.001,E2 -6570.001} C_VEL
LIN {X 0,Y 488.019,Z 402.423,A -85,B 0,C 180,E1 -6570.826,E2 -6570.826} C_VEL
LIN {X 0,Y 488.076,Z 400.708,A -85,B 0,C 180,E1 -6572.477,E2 -6572.477} C_VEL
LIN {X 0,Y 488.108,Z 399.206,A -85,B 0,C 180,E1 -6573.303,E2 -6573.303} C_VEL
LIN {X 0,Y 488.096,Z 396.093,A -85,B 0,C 180,E1 -6574.543,E2 -6574.543} C_VEL
LIN {X 0,Y 488.129,Z 391.874,A -85,B 0,C 180,E1 -6575.785,E2 -6575.785} C_VEL
LIN {X 0,Y 488.195,Z 385.381,A -85,B 0,C 180,E1 -6577.237,E2 -6577.237} C_VEL
LIN {X 0,Y 488.348,Z 378.304,A -85,B 0,C 180,E1 -6578.484,E2 -6578.484} C_VEL
LIN {X 0,Y 488.53,Z 369.405,A -85,B 0,C 180,E1 -6579.733,E2 -6579.733} C_VEL
LIN {X 0,Y 488.856,Z 359.29,A -85,B 0,C 180,E1 -6580.877,E2 -6580.877} C_VEL
LIN {X 0,Y 489.156,Z 348.386,A -85,B 0,C 180,E1 -6581.861,E2 -6581.861} C_VEL
LIN {X 0,Y 489.494,Z 337.559,A -85,B 0,C 180,E1 -6582.649,E2 -6582.649} C_VEL
LIN {X 0,Y 489.841,Z 325.815,A -85,B 0,C 180,E1 -6583.325,E2 -6583.325} C_VEL
LIN {X 0,Y 490.148,Z 312.356,A -85,B 0,C 180,E1 -6583.898,E2 -6583.898} C_VEL
LIN {X 0,Y 490.096,Z 305.534,A -85,B 0,C 180,E1 -6584.124,E2 -6584.124} C_VEL
LIN {X 0,Y 488.968,Z 292.273,A -85,B 0,C 180,E1 -6584.463,E2 -6584.463} C_VEL
LIN {X 0,Y 488.781,Z 290.239,A -85,B 0,C 180,E1 -6584.522,E2 -6584.522} C_VEL
LIN {X 0,Y 489.297,Z 271.13,A -85,B 0,C 180,E1 -6587.773,E2 -6587.773} C_VEL
LIN {X 0,Y 490.108,Z 250.39,A -85,B 0,C 180,E1 -6591.238,E2 -6591.238} C_VEL
LIN {X 0,Y 490.831,Z 232.089,A -85,B 0,C 180,E1 -6594.31,E2 -6594.31} C_VEL
LIN {X 0,Y 491.778,Z 213.575,A -85,B 0,C 180,E1 -6597.504,E2 -6597.504} C_VEL
LIN {X 0,Y 492.542,Z 201.64,A -85,B 0,C 180,E1 -6599.654,E2 -6599.654} C_VEL
LIN {X 0,Y 492.106,Z 197.508,A -85,B 0,C 180,E1 -6600.465,E2 -6600.465} C_VEL
LIN {X 0,Y 489.351,Z 185.472,A -85,B 0,C 180,E1 -6603.077,E2 -6603.077} C_VEL
LIN {X 0,Y 488.711,Z 182.615,A -85,B 0,C 180,E1 -6603.758,E2 -6603.758} C_VEL
LIN {X 0,Y 488.677,Z 182.617,A -85,B 0,C 180,E1 -6606.353,E2 -6606.353} C_VEL
LIN {X 0,Y 488.7,Z 182.61,A -85,B 0,C 180,E1 -6609.255,E2 -6609.255} C_VEL
LIN {X 0,Y 488.712,Z 182.609,A -85,B 0,C 180,E1 -6611.6,E2 -6611.6} C_VEL
LIN {X 0,Y 488.706,Z 182.609,A -85,B 0,C 180,E1 -6614.803,E2 -6614.803} C_VEL
LIN {X 0,Y 488.697,Z 182.614,A -85,B 0,C 180,E1 -6617.475,E2 -6617.475} C_VEL
LIN {X 0,Y 488.738,Z 182.608,A -85,B 0,C 180,E1 -6619.677,E2 -6619.677} C_VEL
LIN {X 0,Y 488.671,Z 182.618,A -85,B 0,C 180,E1 -6622.84,E2 -6622.84} C_VEL
LIN {X 0,Y 488.727,Z 182.741,A -85,B 0,C 180,E1 -6624.76,E2 -6624.76} C_VEL
LIN {X 0,Y 489.226,Z 186.573,A -85,B 0,C 180,E1 -6625.926,E2 -6625.926} C_VEL
LIN {X 0,Y 489.106,Z 196.066,A -85,B 0,C 180,E1 -6628.85,E2 -6628.85} C_VEL
LIN {X 0,Y 489.039,Z 206.336,A -85,B 0,C 180,E1 -6632.156,E2 -6632.156} C_VEL
LIN {X 0,Y 488.956,Z 215.901,A -85,B 0,C 180,E1 -6635.365,E2 -6635.365} C_VEL
LIN {X 0,Y 488.856,Z 224.981,A -85,B 0,C 180,E1 -6638.494,E2 -6638.494} C_VEL
LIN {X 0,Y 488.743,Z 233.908,A -85,B 0,C 180,E1 -6641.636,E2 -6641.636} C_VEL
LIN {X 0,Y 488.634,Z 243.332,A -85,B 0,C 180,E1 -6644.996,E2 -6644.996} C_VEL
LIN {X 0,Y 488.662,Z 244.627,A -85,B 0,C 180,E1 -6645.389,E2 -6645.389} C_VEL
LIN {X 0,Y 490.949,Z 256.312,A -85,B 0,C 180,E1 -6645.783,E2 -6645.783} C_VEL
LIN {X 0,Y 490.608,Z 270.144,A -85,B 0,C 180,E1 -6646.328,E2 -6646.328} C_VEL
LIN {X 0,Y 490.261,Z 282.322,A -85,B 0,C 180,E1 -6646.989,E2 -6646.989} C_VEL
LIN {X 0,Y 489.949,Z 293.683,A -85,B 0,C 180,E1 -6647.785,E2 -6647.785} C_VEL
LIN {X 0,Y 489.507,Z 304.385,A -85,B 0,C 180,E1 -6648.719,E2 -6648.719} C_VEL
LIN {X 0,Y 489.164,Z 313.085,A -85,B 0,C 180,E1 -6649.654,E2 -6649.654} C_VEL
LIN {X 0,Y 488.813,Z 322.523,A -85,B 0,C 180,E1 -6650.9,E2 -6650.9} C_VEL
LIN {X 0,Y 488.506,Z 330.093,A -85,B 0,C 180,E1 -6652.145,E2 -6652.145} C_VEL
LIN {X 0,Y 488.312,Z 336.131,A -85,B 0,C 180,E1 -6653.388,E2 -6653.388} C_VEL
LIN {X 0,Y 488.092,Z 340.907,A -85,B 0,C 180,E1 -6654.63,E2 -6654.63} C_VEL
LIN {X 0,Y 488.125,Z 344.544,A -85,B 0,C 180,E1 -6655.872,E2 -6655.872} C_VEL
LIN {X 0,Y 488.08,Z 346.411,A -85,B 0,C 180,E1 -6656.698,E2 -6656.698} C_VEL
LIN {X 0,Y 488.006,Z 347.851,A -85,B 0,C 180,E1 -6657.524,E2 -6657.524} C_VEL
LIN {X 0,Y 487.846,Z 349.452,A -85,B 0,C 180,E1 -6659.175,E2 -6659.175} C_VEL
LIN {X 0,Y 487.836,Z 349.672,A -85,B 0,C 180,E1 -6660,E2 -6660} C_VEL
LIN {X 0,Y 487.845,Z 349.462,A -85,B 0,C 180,E1 -6660.825,E2 -6660.825} C_VEL
LIN {X 0,Y 488.005,Z 347.836,A -85,B 0,C 180,E1 -6662.476,E2 -6662.476} C_VEL
LIN {X 0,Y 488.066,Z 346.427,A -85,B 0,C 180,E1 -6663.302,E2 -6663.302} C_VEL
LIN {X 0,Y 488.097,Z 343.484,A -85,B 0,C 180,E1 -6664.542,E2 -6664.542} C_VEL
LIN {X 0,Y 488.2,Z 339.493,A -85,B 0,C 180,E1 -6665.784,E2 -6665.784} C_VEL
LIN {X 0,Y 488.353,Z 333.44,A -85,B 0,C 180,E1 -6667.213,E2 -6667.213} C_VEL
LIN {X 0,Y 488.6,Z 326.637,A -85,B 0,C 180,E1 -6668.478,E2 -6668.478} C_VEL
LIN {X 0,Y 488.9,Z 318.268,A -85,B 0,C 180,E1 -6669.724,E2 -6669.724} C_VEL
LIN {X 0,Y 489.184,Z 309.681,A -85,B 0,C 180,E1 -6670.764,E2 -6670.764} C_VEL
LIN {X 0,Y 489.647,Z 299.179,A -85,B 0,C 180,E1 -6671.802,E2 -6671.802} C_VEL
LIN {X 0,Y 489.972,Z 288.301,A -85,B 0,C 180,E1 -6672.664,E2 -6672.664} C_VEL
LIN {X 0,Y 490.326,Z 277.201,A -85,B 0,C 180,E1 -6673.363,E2 -6673.363} C_VEL
LIN {X 0,Y 490.742,Z 264.321,A -85,B 0,C 180,E1 -6673.985,E2 -6673.985} C_VEL
LIN {X 0,Y 490.661,Z 254.489,A -85,B 0,C 180,E1 -6674.345,E2 -6674.345} C_VEL
LIN {X 0,Y 488.445,Z 243.087,A -85,B 0,C 180,E1 -6674.717,E2 -6674.717} C_VEL
LIN {X 0,Y 488.566,Z 235.171,A -85,B 0,C 180,E1 -6677.583,E2 -6677.583} C_VEL
LIN {X 0,Y 488.676,Z 226.323,A -85,B 0,C 180,E1 -6680.801,E2 -6680.801} C_VEL
LIN {X 0,Y 488.816,Z 218.249,A -85,B 0,C 180,E1 -6683.739,E2 -6683.739} C_VEL
LIN {X 0,Y 488.982,Z 209.343,A -85,B 0,C 180,E1 -6686.986,E2 -6686.986} C_VEL
LIN {X 0,Y 489.16,Z 200.541,A -85,B 0,C 180,E1 -6690.19,E2 -6690.19} C_VEL
LIN {X 0,Y 489.289,Z 191.224,A -85,B 0,C 180,E1 -6693.581,E2 -6693.581} C_VEL
LIN {X 0,Y 489.191,Z 185.68,A -85,B 0,C 180,E1 -6695.581,E2 -6695.581} C_VEL
LIN {X 0,Y 488.719,Z 182.611,A -85,B 0,C 180,E1 -6696.736,E2 -6696.736} C_VEL
LIN {X 0,Y 488.705,Z 182.612,A -85,B 0,C 180,E1 -6699.254,E2 -6699.254} C_VEL
LIN {X 0,Y 488.703,Z 182.61,A -85,B 0,C 180,E1 -6701.598,E2 -6701.598} C_VEL
LIN {X 0,Y 488.706,Z 182.608,A -85,B 0,C 180,E1 -6704.802,E2 -6704.802} C_VEL
LIN {X 0,Y 488.697,Z 182.613,A -85,B 0,C 180,E1 -6707.474,E2 -6707.474} C_VEL
LIN {X 0,Y 488.739,Z 182.605,A -85,B 0,C 180,E1 -6709.676,E2 -6709.676} C_VEL
LIN {X 0,Y 488.656,Z 182.617,A -85,B 0,C 180,E1 -6712.838,E2 -6712.838} C_VEL
LIN {X 0,Y 488.725,Z 182.609,A -85,B 0,C 180,E1 -6715.886,E2 -6715.886} C_VEL
LIN {X 0,Y 488.721,Z 182.608,A -85,B 0,C 180,E1 -6717.083,E2 -6717.083} C_VEL
LIN {X 0,Y 488.017,Z 182.696,A -85,B 0,C 180,E1 -6717.771,E2 -6717.771} C_VEL
LIN {X 0,Y 485.114,Z 183.061,A -85,B 0,C 180,E1 -6718.888,E2 -6718.888} C_VEL
LIN {X 0,Y 482.664,Z 183.366,A -85,B 0,C 180,E1 -6719.788,E2 -6719.788} C_VEL
LIN {X 0,Y 481.596,Z 183.499,A -85,B 0,C 180,E1 -6720.483,E2 -6720.483} C_VEL
LIN {X 0,Y 481.5,Z 183.509,A -85,B 0,C 180,E1 -6720.719,E2 -6720.719} C_VEL
LIN {X 0,Y 481.481,Z 183.514,A -85,B 0,C 180,E1 -6721.203,E2 -6721.203} C_VEL
LIN {X 0,Y 481.419,Z 186.761,A -85,B 0,C 180,E1 -6724.026,E2 -6724.026} C_VEL
LIN {X 0,Y 481.345,Z 190.379,A -85,B 0,C 180,E1 -6726.905,E2 -6726.905} C_VEL
LIN {X 0,Y 481.285,Z 193.601,A -85,B 0,C 180,E1 -6729.483,E2 -6729.483} C_VEL
LIN {X 0,Y 481.223,Z 196.987,A -85,B 0,C 180,E1 -6732.139,E2 -6732.139} C_VEL
LIN {X 0,Y 481.201,Z 200.438,A -85,B 0,C 180,E1 -6734.757,E2 -6734.757} C_VEL
LIN {X 0,Y 481.236,Z 205.29,A -85,B 0,C 180,E1 -6738.201,E2 -6738.201} C_VEL
LIN {X 0,Y 481.187,Z 209.424,A -85,B 0,C 180,E1 -6740.846,E2 -6740.846} C_VEL
LIN {X 0,Y 483.001,Z 218.253,A -85,B 0,C 180,E1 -6741.211,E2 -6741.211} C_VEL
LIN {X 0,Y 482.994,Z 226.353,A -85,B 0,C 180,E1 -6741.632,E2 -6741.632} C_VEL
LIN {X 0,Y 482.85,Z 234.363,A -85,B 0,C 180,E1 -6742.204,E2 -6742.204} C_VEL
LIN {X 0,Y 482.631,Z 240.707,A -85,B 0,C 180,E1 -6742.784,E2 -6742.784} C_VEL
LIN {X 0,Y 482.488,Z 245.357,A -85,B 0,C 180,E1 -6743.307,E2 -6743.307} C_VEL
LIN {X 0,Y 482.317,Z 251.356,A -85,B 0,C 180,E1 -6744.145,E2 -6744.145} C_VEL
LIN {X 0,Y 482.063,Z 255.967,A -85,B 0,C 180,E1 -6744.981,E2 -6744.981} C_VEL
LIN {X 0,Y 481.991,Z 259.537,A -85,B 0,C 180,E1 -6745.818,E2 -6745.818} C_VEL
LIN {X 0,Y 481.735,Z 263.376,A -85,B 0,C 180,E1 -6747.072,E2 -6747.072} C_VEL
LIN {X 0,Y 481.586,Z 265.682,A -85,B 0,C 180,E1 -6748.326,E2 -6748.326} C_VEL
LIN {X 0,Y 481.509,Z 266.495,A -85,B 0,C 180,E1 -6749.163,E2 -6749.163} C_VEL
LIN {X 0,Y 481.48,Z 266.778,A -85,B 0,C 180,E1 -6749.999,E2 -6749.999} C_VEL
LIN {X 0,Y 481.501,Z 266.551,A -85,B 0,C 180,E1 -6750.835,E2 -6750.835} C_VEL
LIN {X 0,Y 481.528,Z 265.805,A -85,B 0,C 180,E1 -6751.672,E2 -6751.672} C_VEL
LIN {X 0,Y 481.588,Z 264.493,A -85,B 0,C 180,E1 -6752.508,E2 -6752.508} C_VEL
LIN {X 0,Y 481.906,Z 261.304,A -85,B 0,C 180,E1 -6753.762,E2 -6753.762} C_VEL
LIN {X 0,Y 481.998,Z 258.271,A -85,B 0,C 180,E1 -6754.599,E2 -6754.599} C_VEL
LIN {X 0,Y 482.305,Z 253.154,A -85,B 0,C 180,E1 -6755.644,E2 -6755.644} C_VEL
LIN {X 0,Y 482.492,Z 247.73,A -85,B 0,C 180,E1 -6756.481,E2 -6756.481} C_VEL
LIN {X 0,Y 482.662,Z 240.59,A -85,B 0,C 180,E1 -6757.319,E2 -6757.319} C_VEL
LIN {X 0,Y 482.854,Z 232.856,A -85,B 0,C 180,E1 -6758.014,E2 -6758.014} C_VEL
LIN {X 0,Y 482.996,Z 224.343,A -85,B 0,C 180,E1 -6758.576,E2 -6758.576} C_VEL
LIN {X 0,Y 482.966,Z 217.969,A -85,B 0,C 180,E1 -6758.893,E2 -6758.893} C_VEL
LIN {X 0,Y 481.173,Z 209.299,A -85,B 0,C 180,E1 -6759.271,E2 -6759.271} C_VEL
LIN {X 0,Y 481.245,Z 205.253,A -85,B 0,C 180,E1 -6761.914,E2 -6761.914} C_VEL
